   // --- Status ---
   IF #distance <= #tolerance THEN
       "HMI_Central_Shifter".CS_Status_Auto_Go_to_Des := 2;
   ELSIF #Drive_To_Pos THEN
       "HMI_Central_Shifter".CS_Status_Auto_Go_to_Des := 1;
   ELSE
       "HMI_Central_Shifter".CS_Status_Auto_Go_to_Des := 0;
   END_IF;



   // --- Granice bezpieczeństwa ---
   IF #Actual_Pos <= 0 THEN
       #Auto_Drive_Forward := FALSE;
       #Auto_Drive_Backward := FALSE;
       #Auto_Speed := 0.0;
       #DecelTimer.IN := FALSE;
       #RampActive := FALSE;
       #StopRampTimer.IN := FALSE;
   END_IF;
END_REGION
END_FUNCTION_BLOCK

FUNCTION_BLOCK "CentralShifter_SideShifters"   // FB17, LAD
{ S7_Optimized_Access := 'TRUE' }
// stored: MemoryReserve 100, SetENOAutomatically false
   VAR_INPUT
      In_Side_Drive_Pos : Bool;
      Position_CS : Int;
   END_VAR
   VAR_OUTPUT
      qLeftSide_in_Mid : Bool;
      qRightSide_in_Mid : Bool;
   END_VAR
   VAR
      Side_Hydraulic_CS_RL { S7_SetPoint := 'True'} : "Side_Hydraulic";
      Side_Hydraulic_CS_RR { S7_SetPoint := 'True'} : "Side_Hydraulic";
      Side_Driver_CS { S7_SetPoint := 'True'} : "Side_Driver";
      RL_Speed { S7_SetPoint := 'True'} : Int;
      RP_Speed : Int;
      CentralShifter_Side_Auto_Instance { S7_SetPoint := 'True'} : "CentralShifter_Side_Auto";
      SL_Auto_Speed { S7_SetPoint := 'True'} : Int;
      SR_Auto_Speed : Int;
      SL_Auto_Forward : Bool;
      SL_Auto_Backward : Bool;
      SR_Auto_Forward : Bool;
      SR_Auto_Backward : Bool;
      Sides_In_Position : Bool;
      Sides_In_H3_Pos : Bool;
      Sides_In_H5_Pos : Bool;
      Sides_In_CS_Pos : Bool;
      LightUp : Bool;
      LightMid : Bool;
      LightDown : Bool;
      SR_Error_Laser : Bool;
      SL_Error_Laser : Bool;
      Auto_Position_RL_Up : DInt;
      Auto_Position_RL_Mid : DInt;
      Auto_Position_RL_Down : DInt;
      Auto_Position_RR_Up : DInt;
      Auto_Position_RR_Mid : DInt;
      Auto_Position_RR_Down : DInt;
      Auto_Correction_RR : Int;
   END_VAR
   VAR RETAIN
      Stations : Array[7..13] of "CS_Sides_Stations";
   END_VAR
   VAR
      Status_Side_Go_H3 { S7_SetPoint := 'True'} : Int;
      Status_Side_Go_H5 : Int;
      Status_Side_Go_CS : Int;
      Auto_Hydraulic_Permission_H3 : Bool;
      Auto_Hydraulic_Permission_H5 : Bool;
      Auto_Hydraulic_Up_Timer { S7_SetPoint := 'True'} : TP_TIME;
      Auto_Hydraulic_Down_Timer { S7_SetPoint := 'True'} : TP_TIME;
      Station_H3_Empty : Bool;
      Station_H5_Empty : Bool;
      CS_R1_Sen_Up : Bool;
      CS_R1_Sen_Down : Bool;
      CS_R2_Sen_Up : Bool;
      CS_R2_Sen_Down : Bool;
      Auto_hyd_Up : Bool;
      Auto_hyd_Down : Bool;
      Hyd_Up_Status : Int;
      Hyd_Down_Status : Int;
      CS_RL_Error_Hyd : Bool;
      CS_RR_Error_Hyd : Bool;
      CS_Error_Hyd : Bool;
      CS_Error_Drive : Bool;
   END_VAR
   VAR CONSTANT
      Tolerance : Int := 60;
   END_VAR
   // Stations[7].RL_H3_Pos := 13516;
   // Stations[8].RL_H3_Pos := 13505;
   // Stations[9].RL_H3_Pos := 13520;
   // Stations[10].RL_H3_Pos := 13522;
   // Stations[11].RL_H3_Pos := 13526;
   // Stations[12].RL_H3_Pos := 13505;
   // Stations[13].RL_H3_Pos := 13500;
   // Stations[7].RR_H3_Pos := 13523;
   // Stations[8].RR_H3_Pos := 13495;
   // Stations[9].RR_H3_Pos := 13518;
   // Stations[10].RR_H3_Pos := 13527;
   // Stations[11].RR_H3_Pos := 13524;
   // Stations[12..13].RR_H3_Pos := 13525;
   // Stations[7].RL_Mid_Pos := 7915;
   // Stations[8].RL_Mid_Pos := 7910;
   // Stations[9].RL_Mid_Pos := 7933;
   // Stations[10].RL_Mid_Pos := 7928;
   // Stations[11].RL_Mid_Pos := 7937;
   // Stations[12].RL_Mid_Pos := 7932;
   // Stations[13].RL_Mid_Pos := 7916;
   // Stations[7].RR_Mid_Pos := 7925;
   // Stations[8].RR_Mid_Pos := 7895;
   // Stations[9].RR_Mid_Pos := 7922;
   // Stations[10].RR_Mid_Pos := 7935;
   // Stations[11].RR_Mid_Pos := 7926;
   // Stations[12].RR_Mid_Pos := 7932;
   // Stations[13].RR_Mid_Pos := 7939;
   // Stations[7].RL_H5_Pos := 1930;
   // Stations[8].RL_H5_Pos := 1917;
   // Stations[9].RL_H5_Pos := 1928;
   // Stations[10].RL_H5_Pos := 1929;
   // Stations[11].RL_H5_Pos := 1936;
   // Stations[12].RL_H5_Pos := 1924;
   // Stations[13].RL_H5_Pos := 1918;
   // Stations[7].RR_H5_Pos := 1929;
   // Stations[8].RR_H5_Pos := 1900;
   // Stations[9].RR_H5_Pos := 1921;
   // Stations[10].RR_H5_Pos := 1933;
   // Stations[11].RR_H5_Pos := 1928;
   // Stations[12].RR_H5_Pos := 1934;
   // Stations[13].RR_H5_Pos := 1915;
   // Stations[7].Correction := -20;
   // Stations[8].Correction := -15;
   // Stations[9].Correction := -5;
   // Stations[11].Correction := 0;
   // Stations[12].Correction := 10;
   // Stations[13].Correction := 15;
BEGIN

REGION Network 1: Hydraulic_RL
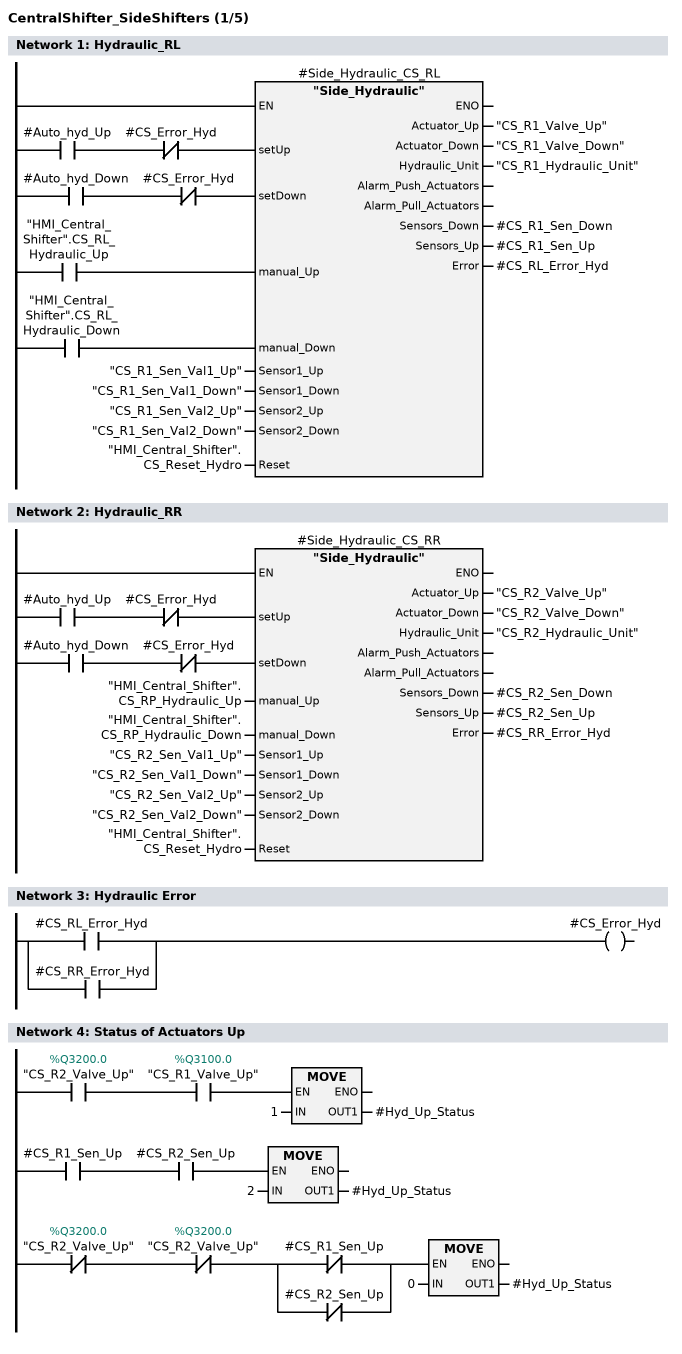
   RUNG wire#powerrail
      #Side_Hydraulic_CS_RL(setUp := wire#w1, setDown := wire#w2, manual_Up := wire#w3, manual_Down := wire#w4, Sensor1_Up := "CS_R1_Sen_Val1_Up", Sensor1_Down := "CS_R1_Sen_Val1_Down", Sensor2_Up := "CS_R1_Sen_Val2_Up", Sensor2_Down := "CS_R1_Sen_Val2_Down", Reset := "HMI_Central_Shifter".CS_Reset_Hydro, Actuator_Up => "CS_R1_Valve_Up", Actuator_Down => "CS_R1_Valve_Down", Hydraulic_Unit => "CS_R1_Hydraulic_Unit", Alarm_Push_Actuators =>, Alarm_Pull_Actuators =>, Sensors_Down => #CS_R1_Sen_Down, Sensors_Up => #CS_R1_Sen_Up, Error => #CS_RL_Error_Hyd)
   END_RUNG
   RUNG wire#powerrail
      Contact( #Auto_hyd_Up )
      I_Contact( #CS_Error_Hyd )
   END_RUNG wire#w1
   RUNG wire#powerrail
      Contact( #Auto_hyd_Down )
      I_Contact( #CS_Error_Hyd )
   END_RUNG wire#w2
   RUNG wire#powerrail
      Contact( "HMI_Central_Shifter".CS_RL_Hydraulic_Up )
   END_RUNG wire#w3
   RUNG wire#powerrail
      Contact( "HMI_Central_Shifter".CS_RL_Hydraulic_Down )
   END_RUNG wire#w4
   // the same network as SCL:
   #Side_Hydraulic_CS_RL(setUp := #Auto_hyd_Up AND NOT #CS_Error_Hyd,   // "Side_Hydraulic"
                         setDown := #Auto_hyd_Down AND NOT #CS_Error_Hyd,
                         manual_Up := "HMI_Central_Shifter".CS_RL_Hydraulic_Up,
                         manual_Down := "HMI_Central_Shifter".CS_RL_Hydraulic_Down,
                         Sensor1_Up := "CS_R1_Sen_Val1_Up",
                         Sensor1_Down := "CS_R1_Sen_Val1_Down",
                         Sensor2_Up := "CS_R1_Sen_Val2_Up",
                         Sensor2_Down := "CS_R1_Sen_Val2_Down",
                         Reset := "HMI_Central_Shifter".CS_Reset_Hydro,
                         Actuator_Up => "CS_R1_Valve_Up",
                         Actuator_Down => "CS_R1_Valve_Down",
                         Hydraulic_Unit => "CS_R1_Hydraulic_Unit",
                         Sensors_Down => #CS_R1_Sen_Down,
                         Sensors_Up => #CS_R1_Sen_Up,
                         Error => #CS_RL_Error_Hyd);
END_REGION

REGION Network 2: Hydraulic_RR
   RUNG wire#powerrail
      #Side_Hydraulic_CS_RR(setUp := wire#w1, setDown := wire#w2, manual_Up := "HMI_Central_Shifter".CS_RP_Hydraulic_Up, manual_Down := "HMI_Central_Shifter".CS_RP_Hydraulic_Down, Sensor1_Up := "CS_R2_Sen_Val1_Up", Sensor1_Down := "CS_R2_Sen_Val1_Down", Sensor2_Up := "CS_R2_Sen_Val2_Up", Sensor2_Down := "CS_R2_Sen_Val2_Down", Reset := "HMI_Central_Shifter".CS_Reset_Hydro, Actuator_Up => "CS_R2_Valve_Up", Actuator_Down => "CS_R2_Valve_Down", Hydraulic_Unit => "CS_R2_Hydraulic_Unit", Alarm_Push_Actuators =>, Alarm_Pull_Actuators =>, Sensors_Down => #CS_R2_Sen_Down, Sensors_Up => #CS_R2_Sen_Up, Error => #CS_RR_Error_Hyd)
   END_RUNG
   RUNG wire#powerrail
      Contact( #Auto_hyd_Up )
      I_Contact( #CS_Error_Hyd )
   END_RUNG wire#w1
   RUNG wire#powerrail
      Contact( #Auto_hyd_Down )
      I_Contact( #CS_Error_Hyd )
   END_RUNG wire#w2
   // the same network as SCL:
   #Side_Hydraulic_CS_RR(setUp := #Auto_hyd_Up AND NOT #CS_Error_Hyd,   // "Side_Hydraulic"
                         setDown := #Auto_hyd_Down AND NOT #CS_Error_Hyd,
                         manual_Up := "HMI_Central_Shifter".CS_RP_Hydraulic_Up,
                         manual_Down := "HMI_Central_Shifter".CS_RP_Hydraulic_Down,
                         Sensor1_Up := "CS_R2_Sen_Val1_Up",
                         Sensor1_Down := "CS_R2_Sen_Val1_Down",
                         Sensor2_Up := "CS_R2_Sen_Val2_Up",
                         Sensor2_Down := "CS_R2_Sen_Val2_Down",
                         Reset := "HMI_Central_Shifter".CS_Reset_Hydro,
                         Actuator_Up => "CS_R2_Valve_Up",
                         Actuator_Down => "CS_R2_Valve_Down",
                         Hydraulic_Unit => "CS_R2_Hydraulic_Unit",
                         Sensors_Down => #CS_R2_Sen_Down,
                         Sensors_Up => #CS_R2_Sen_Up,
                         Error => #CS_RR_Error_Hyd);
END_REGION

REGION Network 3: Hydraulic Error
   RUNG wire#powerrail
      Contact( #CS_RL_Error_Hyd )
      wire#w1
      Coil( #CS_Error_Hyd )
   END_RUNG
   RUNG wire#powerrail
      Contact( #CS_RR_Error_Hyd )
   END_RUNG wire#w1
   // the same network as SCL:
   #CS_Error_Hyd := #CS_RL_Error_Hyd OR #CS_RR_Error_Hyd;
END_REGION

REGION Network 4: Status of Actuators Up
   RUNG wire#powerrail
      Contact( "CS_R2_Valve_Up" )
      Contact( "CS_R1_Valve_Up" )
      Move(in := 1, out1 => #Hyd_Up_Status)
   END_RUNG
   RUNG wire#powerrail
      Contact( #CS_R1_Sen_Up )
      Contact( #CS_R2_Sen_Up )
      Move(in := 2, out1 => #Hyd_Up_Status)
   END_RUNG
   RUNG wire#powerrail
      I_Contact( "CS_R2_Valve_Up" )
      I_Contact( "CS_R2_Valve_Up" )
      wire#w1
      I_Contact( #CS_R1_Sen_Up )
      wire#w2
      Move(in := 0, out1 => #Hyd_Up_Status)
   END_RUNG
   RUNG wire#w1
      I_Contact( #CS_R2_Sen_Up )
   END_RUNG wire#w2
   // the same network as SCL:
   IF "CS_R2_Valve_Up" AND "CS_R1_Valve_Up" THEN #Hyd_Up_Status := 1; END_IF;
   IF #CS_R1_Sen_Up AND #CS_R2_Sen_Up THEN #Hyd_Up_Status := 2; END_IF;
   IF NOT "CS_R2_Valve_Up" AND NOT "CS_R2_Valve_Up" AND (NOT #CS_R1_Sen_Up OR NOT #CS_R2_Sen_Up) THEN
       #Hyd_Up_Status := 0;
   END_IF;
END_REGION

REGION Network 5: Status of Actuators Down
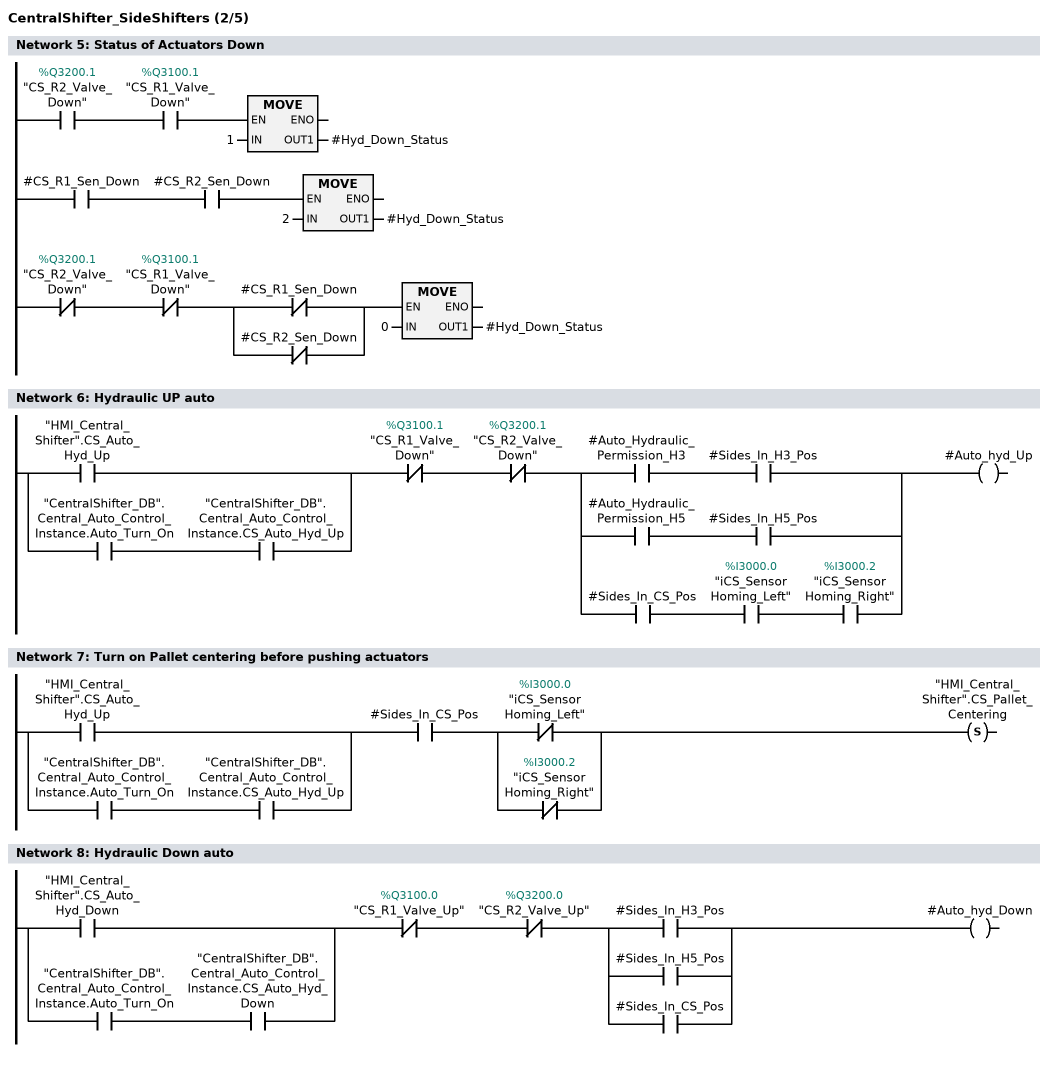
   RUNG wire#powerrail
      Contact( "CS_R2_Valve_Down" )
      Contact( "CS_R1_Valve_Down" )
      Move(in := 1, out1 => #Hyd_Down_Status)
   END_RUNG
   RUNG wire#powerrail
      Contact( #CS_R1_Sen_Down )
      Contact( #CS_R2_Sen_Down )
      Move(in := 2, out1 => #Hyd_Down_Status)
   END_RUNG
   RUNG wire#powerrail
      I_Contact( "CS_R2_Valve_Down" )
      I_Contact( "CS_R1_Valve_Down" )
      wire#w1
      I_Contact( #CS_R1_Sen_Down )
      wire#w2
      Move(in := 0, out1 => #Hyd_Down_Status)
   END_RUNG
   RUNG wire#w1
      I_Contact( #CS_R2_Sen_Down )
   END_RUNG wire#w2
   // the same network as SCL:
   IF "CS_R2_Valve_Down" AND "CS_R1_Valve_Down" THEN #Hyd_Down_Status := 1; END_IF;
   IF #CS_R1_Sen_Down AND #CS_R2_Sen_Down THEN #Hyd_Down_Status := 2; END_IF;
   IF NOT "CS_R2_Valve_Down" AND NOT "CS_R1_Valve_Down" AND (NOT #CS_R1_Sen_Down OR NOT #CS_R2_Sen_Down) THEN
       #Hyd_Down_Status := 0;
   END_IF;
END_REGION

REGION Network 6: Hydraulic UP auto
   RUNG wire#powerrail
      Contact( "HMI_Central_Shifter".CS_Auto_Hyd_Up )
      wire#w1
      I_Contact( "CS_R1_Valve_Down" )
      I_Contact( "CS_R2_Valve_Down" )
      wire#w2
      Contact( #Auto_Hydraulic_Permission_H3 )
      Contact( #Sides_In_H3_Pos )
      wire#w3
      Coil( #Auto_hyd_Up )
   END_RUNG
   RUNG wire#powerrail
      Contact( "CentralShifter_DB".Central_Auto_Control_Instance.Auto_Turn_On )
      Contact( "CentralShifter_DB".Central_Auto_Control_Instance.CS_Auto_Hyd_Up )
   END_RUNG wire#w1
   RUNG wire#w2
      Contact( #Auto_Hydraulic_Permission_H5 )
      Contact( #Sides_In_H5_Pos )
   END_RUNG wire#w3
   RUNG wire#w2
      Contact( #Sides_In_CS_Pos )
      Contact( "iCS_SensorHoming_Left" )
      Contact( "iCS_SensorHoming_Right" )
   END_RUNG wire#w3
   // the same network as SCL:
   #Auto_hyd_Up := ("HMI_Central_Shifter".CS_Auto_Hyd_Up OR ("CentralShifter_DB".Central_Auto_Control_Instance.Auto_Turn_On AND "CentralShifter_DB".Central_Auto_Control_Instance.CS_Auto_Hyd_Up)) AND NOT "CS_R1_Valve_Down" AND NOT "CS_R2_Valve_Down" AND ((#Auto_Hydraulic_Permission_H3 AND #Sides_In_H3_Pos) OR (#Auto_Hydraulic_Permission_H5 AND #Sides_In_H5_Pos) OR (#Sides_In_CS_Pos AND "iCS_SensorHoming_Left" AND "iCS_SensorHoming_Right"));
END_REGION

REGION Network 7: Turn on Pallet centering before pushing actuators
   RUNG wire#powerrail
      Contact( "HMI_Central_Shifter".CS_Auto_Hyd_Up )
      wire#w1
      Contact( #Sides_In_CS_Pos )
      wire#w2
      I_Contact( "iCS_SensorHoming_Left" )
      wire#w3
      S_Coil( "HMI_Central_Shifter".CS_Pallet_Centering )
   END_RUNG
   RUNG wire#powerrail
      Contact( "CentralShifter_DB".Central_Auto_Control_Instance.Auto_Turn_On )
      Contact( "CentralShifter_DB".Central_Auto_Control_Instance.CS_Auto_Hyd_Up )
   END_RUNG wire#w1
   RUNG wire#w2
      I_Contact( "iCS_SensorHoming_Right" )
   END_RUNG wire#w3
   // the same network as SCL:
   IF ("HMI_Central_Shifter".CS_Auto_Hyd_Up OR ("CentralShifter_DB".Central_Auto_Control_Instance.Auto_Turn_On AND "CentralShifter_DB".Central_Auto_Control_Instance.CS_Auto_Hyd_Up)) AND #Sides_In_CS_Pos AND (NOT "iCS_SensorHoming_Left" OR NOT "iCS_SensorHoming_Right") THEN
       "HMI_Central_Shifter".CS_Pallet_Centering := TRUE;
   END_IF;
END_REGION

REGION Network 8: Hydraulic Down auto
   RUNG wire#powerrail
      Contact( "HMI_Central_Shifter".CS_Auto_Hyd_Down )
      wire#w1
      I_Contact( "CS_R1_Valve_Up" )
      I_Contact( "CS_R2_Valve_Up" )
      wire#w2
      Contact( #Sides_In_H3_Pos )
      wire#w3
      Coil( #Auto_hyd_Down )
   END_RUNG
   RUNG wire#powerrail
      Contact( "CentralShifter_DB".Central_Auto_Control_Instance.Auto_Turn_On )
      Contact( "CentralShifter_DB".Central_Auto_Control_Instance.CS_Auto_Hyd_Down )
   END_RUNG wire#w1
   RUNG wire#w2
      Contact( #Sides_In_H5_Pos )
   END_RUNG wire#w3
   RUNG wire#w2
      Contact( #Sides_In_CS_Pos )
   END_RUNG wire#w3
   // the same network as SCL:
   #Auto_hyd_Down := ("HMI_Central_Shifter".CS_Auto_Hyd_Down OR ("CentralShifter_DB".Central_Auto_Control_Instance.Auto_Turn_On AND "CentralShifter_DB".Central_Auto_Control_Instance.CS_Auto_Hyd_Down)) AND NOT "CS_R1_Valve_Up" AND NOT "CS_R2_Valve_Up" AND (#Sides_In_H3_Pos OR #Sides_In_H5_Pos OR #Sides_In_CS_Pos);
END_REGION

REGION Network 9: Laser Error
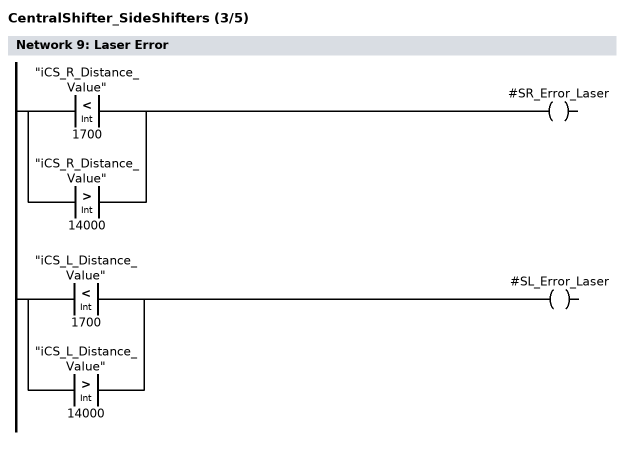
   RUNG wire#powerrail
      { S7_Templates := "SrcType := Int" } LT_Contact(in1 := "iCS_R_Distance_Value", in2 := 1700)
      wire#w1
      Coil( #SR_Error_Laser )
   END_RUNG
   RUNG wire#powerrail
      { S7_Templates := "SrcType := Int" } GT_Contact(in1 := "iCS_R_Distance_Value", in2 := 14000)
   END_RUNG wire#w1
   RUNG wire#powerrail
      { S7_Templates := "SrcType := Int" } LT_Contact(in1 := "iCS_L_Distance_Value", in2 := 1700)
      wire#w2
      Coil( #SL_Error_Laser )
   END_RUNG
   RUNG wire#powerrail
      { S7_Templates := "SrcType := Int" } GT_Contact(in1 := "iCS_L_Distance_Value", in2 := 14000)
   END_RUNG wire#w2
   // the same network as SCL:
   #SR_Error_Laser := ("iCS_R_Distance_Value" < 1700) OR ("iCS_R_Distance_Value" > 14000);
   #SL_Error_Laser := ("iCS_L_Distance_Value" < 1700) OR ("iCS_L_Distance_Value" > 14000);
END_REGION

REGION Network 10 (SCL): Setting SIDE positions by CS_POS
   CASE #Position_CS OF
       7..13:
           #Auto_Position_RL_Up := #Stations[#Position_CS].RL_H3_Pos;
           #Auto_Position_RR_Up := #Stations[#Position_CS].RR_H3_Pos;
           #Auto_Position_RL_Mid := #Stations[#Position_CS].RL_Mid_Pos;
           #Auto_Position_RR_Mid := #Stations[#Position_CS].RR_Mid_Pos;
           #Auto_Position_RL_Down := #Stations[#Position_CS].RL_H5_Pos;
           #Auto_Position_RR_Down := #Stations[#Position_CS].RR_H5_Pos;
           #Auto_Correction_RR := #Stations[#Position_CS].Correction;
       ELSE

           #Auto_Position_RL_Up := 0;
           #Auto_Position_RR_Up := 0;
           #Auto_Position_RL_Mid := 0;
           #Auto_Position_RR_Mid := 0;
           #Auto_Position_RL_Down := 0;
           #Auto_Position_RR_Down := 0;
           #Auto_Correction_RR := 0;
   END_CASE;
END_REGION

REGION Network 11 (SCL): Perform centering during hyd up
   CASE #Position_CS OF
       7..13:
           IF #Sides_In_H3_Pos AND ("HMI_Central_Shifter".CS_Auto_Hyd_Up OR ("CentralShifter_DB".Central_Auto_Control_Instance.Auto_Turn_On AND "CentralShifter_DB".Central_Auto_Control_Instance.CS_Auto_Hyd_Up)) AND NOT "System_To_Moving_Pallets_DB".Centering_Status[#Position_CS, 1] THEN
               "System_To_Moving_Pallets_DB".Centering_Perform[#Position_CS, 1] := 1;
           ELSIF #Sides_In_H5_Pos AND ("HMI_Central_Shifter".CS_Auto_Hyd_Up OR ("CentralShifter_DB".Central_Auto_Control_Instance.Auto_Turn_On AND "CentralShifter_DB".Central_Auto_Control_Instance.CS_Auto_Hyd_Up)) AND NOT "System_To_Moving_Pallets_DB".Centering_Status[#Position_CS, 3] THEN
               "System_To_Moving_Pallets_DB".Centering_Perform[#Position_CS, 3] := 1;
           END_IF;
   END_CASE;
END_REGION

REGION Network 12 (SCL): Permission to hyd up auto
   CASE #Position_CS OF
       7..13:
           IF "System_To_Moving_Pallets_DB".Centering_Status[#Position_CS, 1] THEN

               #Auto_Hydraulic_Permission_H3 := 1;
           ELSE
               #Auto_Hydraulic_Permission_H3 := 0;
           END_IF;

           IF "System_To_Moving_Pallets_DB".Centering_Status[#Position_CS, 3] THEN

               #Auto_Hydraulic_Permission_H5 := 1;
           ELSE
               #Auto_Hydraulic_Permission_H5 := 0;
           END_IF;

   END_CASE;
END_REGION

REGION Network 13 (SCL): Stations empty
   CASE #Position_CS OF
       7..13:
               #Station_H3_Empty := "Pallets_Stations".Stations[4, #Position_CS-3].IsEmpty;

               #Station_H5_Empty := "Pallets_Stations".Stations[2, #Position_CS-2].IsEmpty;

   END_CASE;
END_REGION

REGION Network 14: SIde Drivers
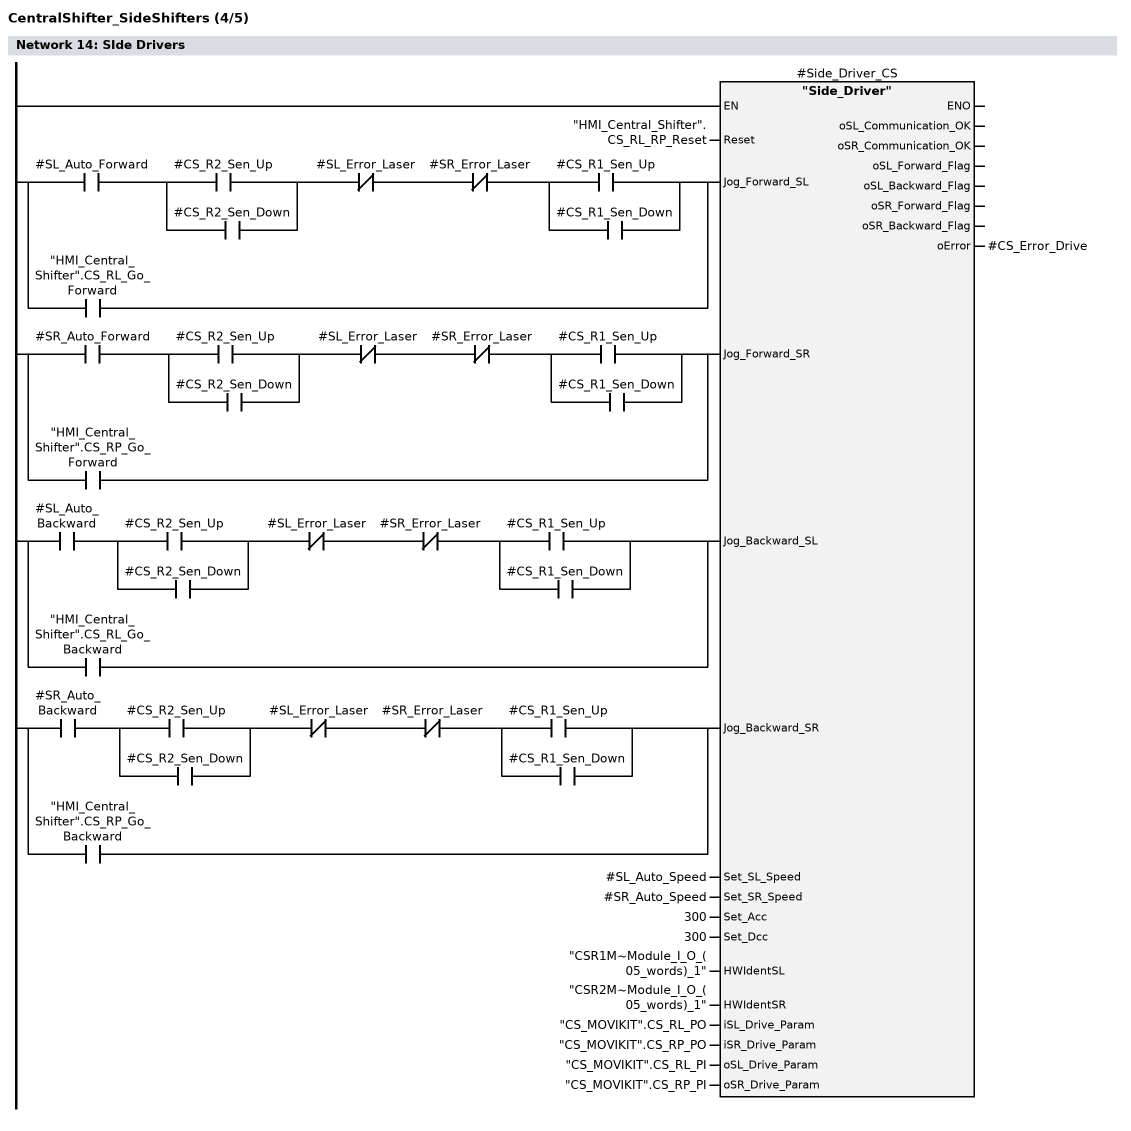
   RUNG wire#powerrail
      #Side_Driver_CS(Jog_Forward_SL := wire#w4, Jog_Forward_SR := wire#w8, Jog_Backward_SL := wire#w12, Jog_Backward_SR := wire#w16, Reset := "HMI_Central_Shifter".CS_RL_RP_Reset, Set_SL_Speed := #SL_Auto_Speed, Set_SR_Speed := #SR_Auto_Speed, Set_Acc := 300, Set_Dcc := 300, HWIdentSL := "CSR1M~Module_I_O_(05_words)_1", HWIdentSR := "CSR2M~Module_I_O_(05_words)_1", iSL_Drive_Param := "CS_MOVIKIT".CS_RL_PO, iSR_Drive_Param := "CS_MOVIKIT".CS_RP_PO, oSL_Drive_Param := "CS_MOVIKIT".CS_RL_PI, oSR_Drive_Param := "CS_MOVIKIT".CS_RP_PI, oSL_Communication_OK =>, oSR_Communication_OK =>, oSL_Forward_Flag =>, oSL_Backward_Flag =>, oSR_Forward_Flag =>, oSR_Backward_Flag =>, oError => #CS_Error_Drive)
   END_RUNG
   RUNG wire#powerrail
      Contact( #SL_Auto_Forward )
      wire#w1
      Contact( #CS_R2_Sen_Up )
      wire#w2
      I_Contact( #SL_Error_Laser )
      I_Contact( #SR_Error_Laser )
      wire#w3
      Contact( #CS_R1_Sen_Up )
   END_RUNG wire#w4
   RUNG wire#w1
      Contact( #CS_R2_Sen_Down )
   END_RUNG wire#w2
   RUNG wire#w3
      Contact( #CS_R1_Sen_Down )
   END_RUNG wire#w4
   RUNG wire#powerrail
      Contact( "HMI_Central_Shifter".CS_RL_Go_Forward )
   END_RUNG wire#w4
   RUNG wire#powerrail
      Contact( #SR_Auto_Forward )
      wire#w5
      Contact( #CS_R2_Sen_Up )
      wire#w6
      I_Contact( #SL_Error_Laser )
      I_Contact( #SR_Error_Laser )
      wire#w7
      Contact( #CS_R1_Sen_Up )
   END_RUNG wire#w8
   RUNG wire#w5
      Contact( #CS_R2_Sen_Down )
   END_RUNG wire#w6
   RUNG wire#w7
      Contact( #CS_R1_Sen_Down )
   END_RUNG wire#w8
   RUNG wire#powerrail
      Contact( "HMI_Central_Shifter".CS_RP_Go_Forward )
   END_RUNG wire#w8
   RUNG wire#powerrail
      Contact( #SL_Auto_Backward )
      wire#w9
      Contact( #CS_R2_Sen_Up )
      wire#w10
      I_Contact( #SL_Error_Laser )
      I_Contact( #SR_Error_Laser )
      wire#w11
      Contact( #CS_R1_Sen_Up )
   END_RUNG wire#w12
   RUNG wire#w9
      Contact( #CS_R2_Sen_Down )
   END_RUNG wire#w10
   RUNG wire#w11
      Contact( #CS_R1_Sen_Down )
   END_RUNG wire#w12
   RUNG wire#powerrail
      Contact( "HMI_Central_Shifter".CS_RL_Go_Backward )
   END_RUNG wire#w12
   RUNG wire#powerrail
      Contact( #SR_Auto_Backward )
      wire#w13
      Contact( #CS_R2_Sen_Up )
      wire#w14
      I_Contact( #SL_Error_Laser )
      I_Contact( #SR_Error_Laser )
      wire#w15
      Contact( #CS_R1_Sen_Up )
   END_RUNG wire#w16
   RUNG wire#w13
      Contact( #CS_R2_Sen_Down )
   END_RUNG wire#w14
   RUNG wire#w15
      Contact( #CS_R1_Sen_Down )
   END_RUNG wire#w16
   RUNG wire#powerrail
      Contact( "HMI_Central_Shifter".CS_RP_Go_Backward )
   END_RUNG wire#w16
   // the same network as SCL:
   #Side_Driver_CS(Reset := "HMI_Central_Shifter".CS_RL_RP_Reset,   // "Side_Driver"
                   Jog_Forward_SL := (#SL_Auto_Forward AND (#CS_R2_Sen_Up OR #CS_R2_Sen_Down) AND NOT #SL_Error_Laser AND NOT #SR_Error_Laser AND (#CS_R1_Sen_Up OR #CS_R1_Sen_Down)) OR "HMI_Central_Shifter".CS_RL_Go_Forward,
                   Jog_Forward_SR := (#SR_Auto_Forward AND (#CS_R2_Sen_Up OR #CS_R2_Sen_Down) AND NOT #SL_Error_Laser AND NOT #SR_Error_Laser AND (#CS_R1_Sen_Up OR #CS_R1_Sen_Down)) OR "HMI_Central_Shifter".CS_RP_Go_Forward,
                   Jog_Backward_SL := (#SL_Auto_Backward AND (#CS_R2_Sen_Up OR #CS_R2_Sen_Down) AND NOT #SL_Error_Laser AND NOT #SR_Error_Laser AND (#CS_R1_Sen_Up OR #CS_R1_Sen_Down)) OR "HMI_Central_Shifter".CS_RL_Go_Backward,
                   Jog_Backward_SR := (#SR_Auto_Backward AND (#CS_R2_Sen_Up OR #CS_R2_Sen_Down) AND NOT #SL_Error_Laser AND NOT #SR_Error_Laser AND (#CS_R1_Sen_Up OR #CS_R1_Sen_Down)) OR "HMI_Central_Shifter".CS_RP_Go_Backward,
                   Set_SL_Speed := #SL_Auto_Speed,
                   Set_SR_Speed := #SR_Auto_Speed,
                   Set_Acc := 300,
                   Set_Dcc := 300,
                   HWIdentSL := "CSR1M~Module_I_O_(05_words)_1",
                   HWIdentSR := "CSR2M~Module_I_O_(05_words)_1",
                   iSL_Drive_Param := "CS_MOVIKIT".CS_RL_PO,
                   iSR_Drive_Param := "CS_MOVIKIT".CS_RP_PO,
                   oSL_Drive_Param := "CS_MOVIKIT".CS_RL_PI,
                   oSR_Drive_Param := "CS_MOVIKIT".CS_RP_PI,
                   oError => #CS_Error_Drive);
END_REGION

REGION Network 15 (SCL): Limit positions of Sides
   IF #Auto_Position_RL_Down > 14000 THEN
       #Auto_Position_RL_Down := 14000;
   ELSIF #Auto_Position_RL_Down < 1800 THEN
       #Auto_Position_RL_Down := 1800;
   END_IF;

   IF #Auto_Position_RL_Up > 14000 THEN
       #Auto_Position_RL_Up := 14000;
   ELSIF #Auto_Position_RL_Up < 1800 THEN
       #Auto_Position_RL_Up := 1800;
   END_IF;

   IF #Auto_Position_RR_Down > 14000 THEN
       #Auto_Position_RR_Down := 14000;
   ELSIF #Auto_Position_RR_Down < 1800 THEN
       #Auto_Position_RR_Down := 1800;
   END_IF;

   IF #Auto_Position_RR_Up > 14000 THEN
       #Auto_Position_RR_Up := 14000;
   ELSIF #Auto_Position_RR_Up < 1800 THEN
       #Auto_Position_RR_Up := 1800;
   END_IF;
END_REGION

REGION Network 16: CS Side Auto
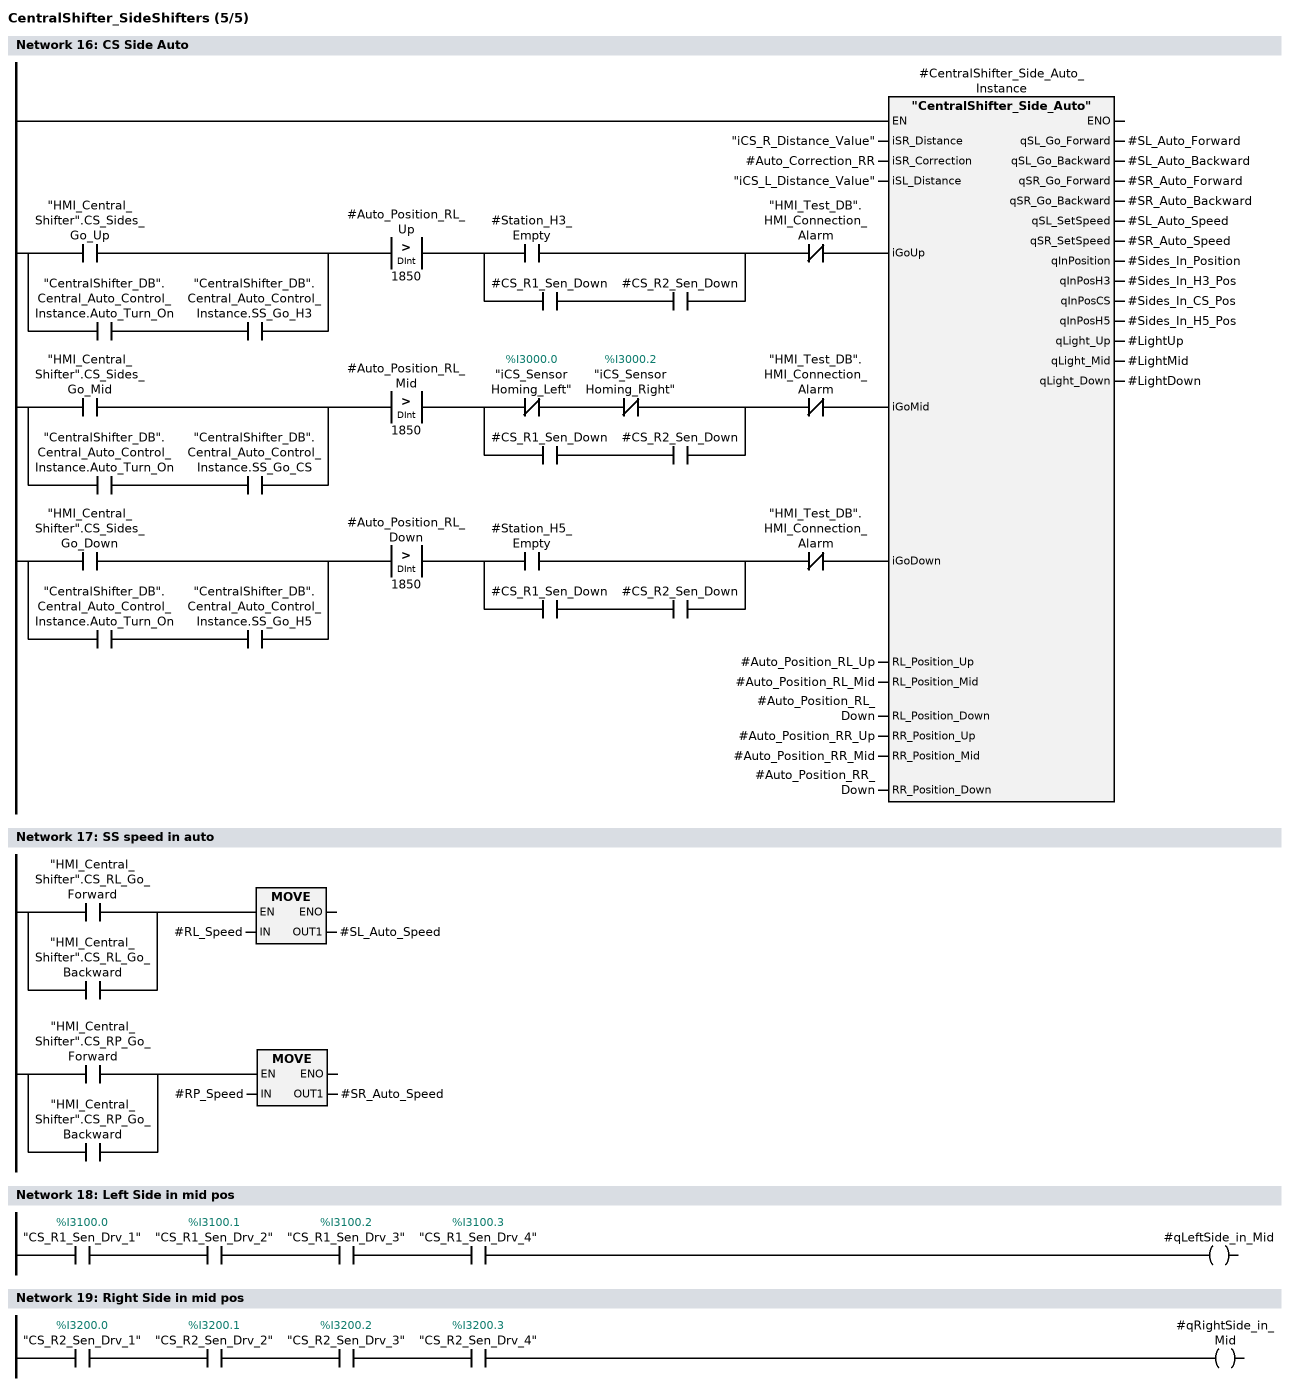
   RUNG wire#powerrail
      #CentralShifter_Side_Auto_Instance(iGoUp := wire#w4, iGoMid := wire#w8, iGoDown := wire#w12, iSR_Distance := "iCS_R_Distance_Value", iSR_Correction := #Auto_Correction_RR, iSL_Distance := "iCS_L_Distance_Value", RL_Position_Up := #Auto_Position_RL_Up, RL_Position_Mid := #Auto_Position_RL_Mid, RL_Position_Down := #Auto_Position_RL_Down, RR_Position_Up := #Auto_Position_RR_Up, RR_Position_Mid := #Auto_Position_RR_Mid, RR_Position_Down := #Auto_Position_RR_Down, qSL_Go_Forward => #SL_Auto_Forward, qSL_Go_Backward => #SL_Auto_Backward, qSR_Go_Forward => #SR_Auto_Forward, qSR_Go_Backward => #SR_Auto_Backward, qSL_SetSpeed => #SL_Auto_Speed, qSR_SetSpeed => #SR_Auto_Speed, qInPosition => #Sides_In_Position, qInPosH3 => #Sides_In_H3_Pos, qInPosCS => #Sides_In_CS_Pos, qInPosH5 => #Sides_In_H5_Pos, qLight_Up => #LightUp, qLight_Mid => #LightMid, qLight_Down => #LightDown)
   END_RUNG
   RUNG wire#powerrail
      Contact( "HMI_Central_Shifter".CS_Sides_Go_Up )
      wire#w1
      { S7_Templates := "SrcType := DInt" } GT_Contact(in1 := #Auto_Position_RL_Up, in2 := 1850)
      wire#w2
      Contact( #Station_H3_Empty )
      wire#w3
      I_Contact( "HMI_Test_DB".HMI_Connection_Alarm )
   END_RUNG wire#w4
   RUNG wire#powerrail
      Contact( "CentralShifter_DB".Central_Auto_Control_Instance.Auto_Turn_On )
      Contact( "CentralShifter_DB".Central_Auto_Control_Instance.SS_Go_H3 )
   END_RUNG wire#w1
   RUNG wire#w2
      Contact( #CS_R1_Sen_Down )
      Contact( #CS_R2_Sen_Down )
   END_RUNG wire#w3
   RUNG wire#powerrail
      Contact( "HMI_Central_Shifter".CS_Sides_Go_Mid )
      wire#w5
      { S7_Templates := "SrcType := DInt" } GT_Contact(in1 := #Auto_Position_RL_Mid, in2 := 1850)
      wire#w6
      I_Contact( "iCS_SensorHoming_Left" )
      I_Contact( "iCS_SensorHoming_Right" )
      wire#w7
      I_Contact( "HMI_Test_DB".HMI_Connection_Alarm )
   END_RUNG wire#w8
   RUNG wire#powerrail
      Contact( "CentralShifter_DB".Central_Auto_Control_Instance.Auto_Turn_On )
      Contact( "CentralShifter_DB".Central_Auto_Control_Instance.SS_Go_CS )
   END_RUNG wire#w5
   RUNG wire#w6
      Contact( #CS_R1_Sen_Down )
      Contact( #CS_R2_Sen_Down )
   END_RUNG wire#w7
   RUNG wire#powerrail
      Contact( "HMI_Central_Shifter".CS_Sides_Go_Down )
      wire#w9
      { S7_Templates := "SrcType := DInt" } GT_Contact(in1 := #Auto_Position_RL_Down, in2 := 1850)
      wire#w10
      Contact( #Station_H5_Empty )
      wire#w11
      I_Contact( "HMI_Test_DB".HMI_Connection_Alarm )
   END_RUNG wire#w12
   RUNG wire#powerrail
      Contact( "CentralShifter_DB".Central_Auto_Control_Instance.Auto_Turn_On )
      Contact( "CentralShifter_DB".Central_Auto_Control_Instance.SS_Go_H5 )
   END_RUNG wire#w9
   RUNG wire#w10
      Contact( #CS_R1_Sen_Down )
      Contact( #CS_R2_Sen_Down )
   END_RUNG wire#w11
   // the same network as SCL:
   #CentralShifter_Side_Auto_Instance(iSR_Distance := "iCS_R_Distance_Value",   // "CentralShifter_Side_Auto"
                           iSR_Correction := #Auto_Correction_RR,
                           iSL_Distance := "iCS_L_Distance_Value",
                           iGoUp := ("HMI_Central_Shifter".CS_Sides_Go_Up OR ("CentralShifter_DB".Central_Auto_Control_Instance.Auto_Turn_On AND "CentralShifter_DB".Central_Auto_Control_Instance.SS_Go_H3)) AND (#Auto_Position_RL_Up > 1850) AND (#Station_H3_Empty OR (#CS_R1_Sen_Down AND #CS_R2_Sen_Down)) AND NOT "HMI_Test_DB".HMI_Connection_Alarm,
                           iGoMid := ("HMI_Central_Shifter".CS_Sides_Go_Mid OR ("CentralShifter_DB".Central_Auto_Control_Instance.Auto_Turn_On AND "CentralShifter_DB".Central_Auto_Control_Instance.SS_Go_CS)) AND (#Auto_Position_RL_Mid > 1850) AND ((NOT "iCS_SensorHoming_Left" AND NOT "iCS_SensorHoming_Right") OR (#CS_R1_Sen_Down AND #CS_R2_Sen_Down)) AND NOT "HMI_Test_DB".HMI_Connection_Alarm,
                           iGoDown := ("HMI_Central_Shifter".CS_Sides_Go_Down OR ("CentralShifter_DB".Central_Auto_Control_Instance.Auto_Turn_On AND "CentralShifter_DB".Central_Auto_Control_Instance.SS_Go_H5)) AND (#Auto_Position_RL_Down > 1850) AND (#Station_H5_Empty OR (#CS_R1_Sen_Down AND #CS_R2_Sen_Down)) AND NOT "HMI_Test_DB".HMI_Connection_Alarm,
                           RL_Position_Up := #Auto_Position_RL_Up,
                           RL_Position_Mid := #Auto_Position_RL_Mid,
                           RL_Position_Down := #Auto_Position_RL_Down,
                           RR_Position_Up := #Auto_Position_RR_Up,
                           RR_Position_Mid := #Auto_Position_RR_Mid,
                           RR_Position_Down := #Auto_Position_RR_Down,
                           qSL_Go_Forward => #SL_Auto_Forward,
                           qSL_Go_Backward => #SL_Auto_Backward,
                           qSR_Go_Forward => #SR_Auto_Forward,
                           qSR_Go_Backward => #SR_Auto_Backward,
                           qSL_SetSpeed => #SL_Auto_Speed,
                           qSR_SetSpeed => #SR_Auto_Speed,
                           qInPosition => #Sides_In_Position,
                           qInPosH3 => #Sides_In_H3_Pos,
                           qInPosCS => #Sides_In_CS_Pos,
                           qInPosH5 => #Sides_In_H5_Pos,
                           qLight_Up => #LightUp,
                           qLight_Mid => #LightMid,
                           qLight_Down => #LightDown);
END_REGION

REGION Network 17: SS speed in auto
   RUNG wire#powerrail
      Contact( "HMI_Central_Shifter".CS_RL_Go_Forward )
      wire#w1
      Move(in := #RL_Speed, out1 => #SL_Auto_Speed)
   END_RUNG
   RUNG wire#powerrail
      Contact( "HMI_Central_Shifter".CS_RL_Go_Backward )
   END_RUNG wire#w1
   RUNG wire#powerrail
      Contact( "HMI_Central_Shifter".CS_RP_Go_Forward )
      wire#w2
      Move(in := #RP_Speed, out1 => #SR_Auto_Speed)
   END_RUNG
   RUNG wire#powerrail
      Contact( "HMI_Central_Shifter".CS_RP_Go_Backward )
   END_RUNG wire#w2
   // the same network as SCL:
   IF "HMI_Central_Shifter".CS_RL_Go_Forward OR "HMI_Central_Shifter".CS_RL_Go_Backward THEN
       #SL_Auto_Speed := #RL_Speed;
   END_IF;
   IF "HMI_Central_Shifter".CS_RP_Go_Forward OR "HMI_Central_Shifter".CS_RP_Go_Backward THEN
       #SR_Auto_Speed := #RP_Speed;
   END_IF;
END_REGION

REGION Network 18: Left Side in mid pos
   RUNG wire#powerrail
      Contact( "CS_R1_Sen_Drv_1" )
      Contact( "CS_R1_Sen_Drv_2" )
      Contact( "CS_R1_Sen_Drv_3" )
      Contact( "CS_R1_Sen_Drv_4" )
      Coil( #qLeftSide_in_Mid )
   END_RUNG
   // the same network as SCL:
   #qLeftSide_in_Mid := "CS_R1_Sen_Drv_1" AND "CS_R1_Sen_Drv_2" AND "CS_R1_Sen_Drv_3" AND "CS_R1_Sen_Drv_4";
END_REGION

REGION Network 19: Right Side in mid pos
   RUNG wire#powerrail
      Contact( "CS_R2_Sen_Drv_1" )
      Contact( "CS_R2_Sen_Drv_2" )
      Contact( "CS_R2_Sen_Drv_3" )
      Contact( "CS_R2_Sen_Drv_4" )
      Coil( #qRightSide_in_Mid )
   END_RUNG
   // the same network as SCL:
   #qRightSide_in_Mid := "CS_R2_Sen_Drv_1" AND "CS_R2_Sen_Drv_2" AND "CS_R2_Sen_Drv_3" AND "CS_R2_Sen_Drv_4";
END_REGION

REGION Network 20 (SCL): Status - go to destinations
           IF "HMI_Central_Shifter".CS_Sides_Go_Up AND NOT #Sides_In_H3_Pos AND #In_Side_Drive_Pos THEN
               #Status_Side_Go_H3 := 1;
           ELSIF #Sides_In_H3_Pos THEN
               #Status_Side_Go_H3 := 2;
           ELSE
               #Status_Side_Go_H3 := 0;
           END_IF;

           IF "HMI_Central_Shifter".CS_Sides_Go_Down AND NOT #Sides_In_H5_Pos AND #In_Side_Drive_Pos THEN
               #Status_Side_Go_H5 := 1;
           ELSIF #Sides_In_H5_Pos THEN
               #Status_Side_Go_H5 := 2;
           ELSE
               #Status_Side_Go_H5 := 0;
           END_IF;

           IF "HMI_Central_Shifter".CS_Sides_Go_Mid AND NOT #Sides_In_CS_Pos AND #In_Side_Drive_Pos THEN
               #Status_Side_Go_CS := 1;
           ELSIF #Sides_In_CS_Pos THEN
               #Status_Side_Go_CS := 2;
           ELSE
               #Status_Side_Go_CS := 0;
           END_IF;
END_REGION
END_FUNCTION_BLOCK

FUNCTION_BLOCK "CentralShifter_Side_Auto"
{ S7_Optimized_Access := 'TRUE' }
VERSION : 0.1
   VAR_INPUT 
      iSR_Distance : Int;
      iSR_Correction : Int;
      iSL_Distance : Int;
      iGoUp : Bool;
      iGoMid : Bool;
      iGoDown : Bool;
      RL_Position_Up : DInt;
      RL_Position_Mid : DInt;
      RL_Position_Down : DInt;
      RR_Position_Up : DInt;
      RR_Position_Mid : DInt;
      RR_Position_Down : DInt;
   END_VAR

   VAR_OUTPUT 
      qSL_Go_Forward : Bool;
      qSL_Go_Backward : Bool;
      qSR_Go_Forward : Bool;
      qSR_Go_Backward : Bool;
      qSL_SetSpeed : Int;
      qSR_SetSpeed : Int;
      qInPosition : Bool;
      qInPosH3 : Bool;
      qInPosCS : Bool;
      qInPosH5 : Bool;
      qLight_Up : Bool;
      qLight_Mid : Bool;
      qLight_Down : Bool;
   END_VAR

   VAR 
      distanceSL_SR : DInt;
      SR_Correct_Distance : DInt;
      moveActive : Bool;
      targetPosRL : DInt;
      targetPosRR : DInt;
      distanceToTargetSL : DInt;
      distanceToTargetSR : DInt;
      Delta : Real;
   END_VAR

   VAR CONSTANT 
      Tolerance : Int := 2;
      Tolerance_Hydro : Int := 7;
      Tolerance_Light : Int := 10;
      DistanceSlowZone : Int := 300;
      K : Real := 1.5;
      Tolerance_CS : Int := 25;
   END_VAR


BEGIN
	// Reset komend ruchu
	#qSL_Go_Forward := FALSE;
	#qSL_Go_Backward := FALSE;
	#qSR_Go_Forward := FALSE;
	#qSR_Go_Backward := FALSE;
	
	#SR_Correct_Distance := #iSR_Correction + #iSR_Distance;
	#distanceSL_SR := #SR_Correct_Distance - #iSL_Distance;
	
	
	// --- Miganie tylko gdy przycisk TRZYMANY i moveActive ---
	IF #moveActive AND "Clock_2Hz" THEN
	    IF #iGoDown THEN
	        #qLight_Down := 1;
	    ELSE
	        #qLight_Down := 0;
	    END_IF;
	    IF #iGoMid THEN
	        #qLight_Mid := 1;
	    ELSE
	        #qLight_Mid := 0;
	    END_IF;
	    IF #iGoUp THEN
	        #qLight_Up := 1;
	    ELSE
	        #qLight_Up := 0;
	    END_IF;
	ELSE
	    // Gdy nie ma ruchu — zgaś lampki
	    #qLight_Down:= 0;
	    #qLight_Mid := 0;
	    #qLight_Up := 0;
	END_IF;
	
	
	// --- Obsługa dynamicznego wyboru celu ---
	IF #iGoUp THEN
	    #targetPosRL := #RL_Position_Up;
	    #targetPosRR := #RR_Position_Up;
	    #moveActive := TRUE;
	ELSIF #iGoMid THEN
	    #targetPosRL := #RL_Position_Mid;
	    #targetPosRR := #RR_Position_Mid;
	    #moveActive := TRUE;
	ELSIF #iGoDown THEN
	    #targetPosRL := #RL_Position_Down;
	    #targetPosRR := #RR_Position_Down;
	    #moveActive := TRUE;
	ELSE
	    // Żaden przycisk nie trzymany — przerwij ruch
	    #moveActive := FALSE;
	END_IF;
	
	IF NOT "Data_From_Safety".Safety_Active THEN
	    #moveActive := 0;
	    ;
	END_IF;
	
	// --- Jeśli ruch aktywny ---
	IF #moveActive THEN
	    // --- SL (główny) ---
	    #distanceToTargetSL := ABS(#iSL_Distance - #targetPosRL);
	    #distanceToTargetSR := ABS(#SR_Correct_Distance - #targetPosRR);
	    
	    IF #distanceToTargetSL > #Tolerance THEN
	        IF #iSL_Distance > #targetPosRL THEN
	            #qSL_Go_Forward := FALSE;
	            #qSL_Go_Backward := TRUE;
	        ELSE
	            #qSL_Go_Forward := TRUE;
	            #qSL_Go_Backward := FALSE;
	        END_IF;
	        
	        IF #distanceToTargetSL <= #DistanceSlowZone THEN
	            #qSL_SetSpeed := 300;
	        ELSE
	            #qSL_SetSpeed := 1000;
	        END_IF;
	        
	    ELSE
	        #qSL_Go_Forward := FALSE;
	        #qSL_Go_Backward := FALSE;
	        #qSL_SetSpeed := 0;
	        #moveActive := FALSE;
	    END_IF;
	    
	    // --- SR (podąża) ---
	    #distanceSL_SR := #SR_Correct_Distance - #iSL_Distance;
	    //#absDelta := ABS(#distanceSL_SR);
	    // IF #distanceToTargetSL > #Tolerance THEN
	    
	    IF #distanceToTargetSR > #Tolerance THEN
	        IF #SR_Correct_Distance > #targetPosRR THEN
	            #qSR_Go_Forward := FALSE;
	            #qSR_Go_Backward := TRUE;
	        ELSE
	            #qSR_Go_Forward := TRUE;
	            #qSR_Go_Backward := FALSE;
	        END_IF;
	    END_IF;
	    
	    // Kierunek SR = kierunek SL
	    // #qSR_Go_Forward := #qSL_Go_Forward;
	    //#qSR_Go_Backward := #qSL_Go_Backward;
	    
	    // Korekcja prędkości
	    #Delta := #distanceSL_SR * #K;
	    IF #Delta > 1000 THEN
	        #Delta := 1000;
	    ELSIF #Delta < -1000 THEN
	        #Delta := -1000;
	    END_IF;
	    //zamien znaki
	    IF #qSR_Go_Forward THEN
	        #qSR_SetSpeed := #qSL_SetSpeed - #Delta;
	    ELSIF #qSR_Go_Backward THEN
	        #qSR_SetSpeed := #qSL_SetSpeed + #Delta;
	    END_IF;
	    
	    // Ograniczenia
	    IF #qSR_SetSpeed > 1500 THEN
	        #qSR_SetSpeed := 1500;
	    ELSIF #qSR_SetSpeed < 200 THEN
	        #qSR_SetSpeed := 200;
	    END_IF;
	    
	    // END_IF;
	END_IF;
	
	#qInPosition := FALSE;
	#qInPosH3 := FALSE;
	#qInPosCS := FALSE;
	#qInPosH5 := FALSE;
	
	// dolna
	IF (ABS(#iSL_Distance - #RL_Position_Down) <= #Tolerance_Hydro AND ABS(#SR_Correct_Distance - #RR_Position_Down) <= #Tolerance_Hydro) THEN
	    #qInPosition := TRUE;
	    #qInPosH5 := TRUE;
	    
	// cs
	ELSIF (ABS(#iSL_Distance - #RL_Position_Mid) <= #Tolerance_Hydro AND ABS(#SR_Correct_Distance - #RR_Position_Mid) <= #Tolerance_Hydro) THEN
	    #qInPosition := TRUE;
	    #qInPosCS := TRUE;
	    
	// górna
	ELSIF (ABS(#iSL_Distance - #RL_Position_Up) <= #Tolerance_Hydro AND ABS(#SR_Correct_Distance - #RR_Position_Up) <= #Tolerance_Hydro) THEN
	    #qInPosition := TRUE;
	    #qInPosH3 := TRUE;
	END_IF;
	
	
	
	IF (ABS(#iSL_Distance - #RL_Position_Down) <= #Tolerance_Light AND ABS(#SR_Correct_Distance - #RL_Position_Down) <= #Tolerance_Light) THEN
	    #qLight_Down := 1;
	ELSIF (ABS(#iSL_Distance - #RL_Position_Mid) <= #Tolerance_Light AND ABS(#SR_Correct_Distance - #RL_Position_Mid) <= #Tolerance_Light) THEN
	    #qLight_Mid := 1;
	ELSIF (ABS(#iSL_Distance - #RL_Position_Up) <= #Tolerance_Light AND ABS(#SR_Correct_Distance - #RL_Position_Up) <= #Tolerance_Light) THEN
	    #qLight_Up := 1;
	END_IF;
	
END_FUNCTION_BLOCK

FUNCTION_BLOCK "CentralShifter_Move_Pallets"   // FB19, LAD
{ S7_Optimized_Access := 'TRUE' }
// stored: MemoryReserve 100, SetENOAutomatically false
   VAR
      Motor_Driver_Instance { S7_SetPoint := 'True'} : "Side_Driver";
      Speed : Int := 400;
      Auto_Go_Left : Bool;
      Auto_Go_Right : Bool;
      CSM1_Comm_ok : Bool;
      CSM2_Comm_ok : Bool;
      prevCentering : Bool;
      tCenteringTimer : TON_TIME;
   END_VAR
   VAR_TEMP
      "czujnik lewy" : Bool;
      "czujnik prawy" : Bool;
   END_VAR
BEGIN

REGION Network 1
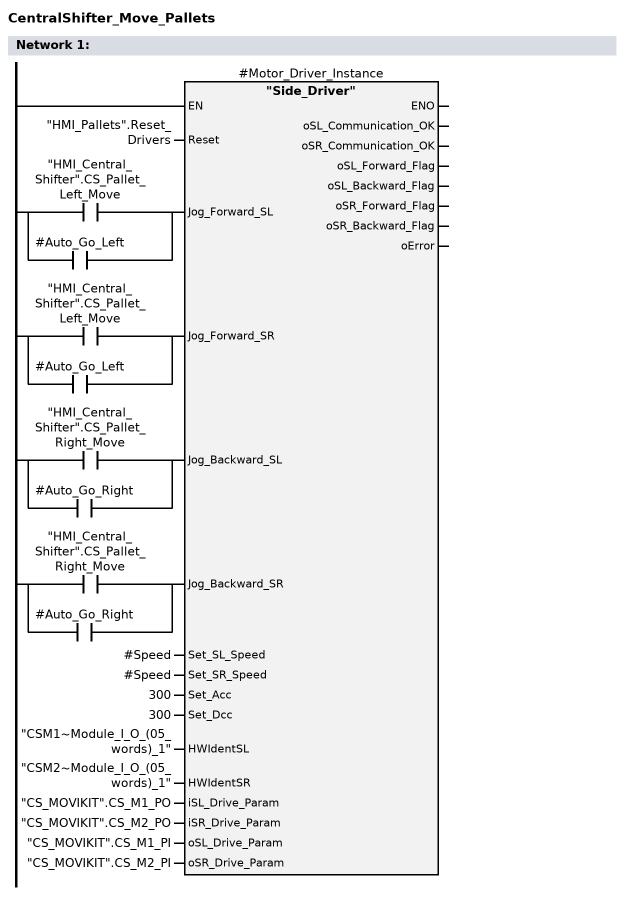
   RUNG wire#powerrail
      #Motor_Driver_Instance(Jog_Forward_SL := wire#w1, Jog_Forward_SR := wire#w2, Jog_Backward_SL := wire#w3, Jog_Backward_SR := wire#w4, Reset := "HMI_Pallets".Reset_Drivers, Set_SL_Speed := #Speed, Set_SR_Speed := #Speed, Set_Acc := 300, Set_Dcc := 300, HWIdentSL := "CSM1~Module_I_O_(05_words)_1", HWIdentSR := "CSM2~Module_I_O_(05_words)_1", iSL_Drive_Param := "CS_MOVIKIT".CS_M1_PO, iSR_Drive_Param := "CS_MOVIKIT".CS_M2_PO, oSL_Drive_Param := "CS_MOVIKIT".CS_M1_PI, oSR_Drive_Param := "CS_MOVIKIT".CS_M2_PI, oSL_Communication_OK =>, oSR_Communication_OK =>, oSL_Forward_Flag =>, oSL_Backward_Flag =>, oSR_Forward_Flag =>, oSR_Backward_Flag =>, oError =>)
   END_RUNG
   RUNG wire#powerrail
      Contact( "HMI_Central_Shifter".CS_Pallet_Left_Move )
   END_RUNG wire#w1
   RUNG wire#powerrail
      Contact( #Auto_Go_Left )
   END_RUNG wire#w1
   RUNG wire#powerrail
      Contact( "HMI_Central_Shifter".CS_Pallet_Left_Move )
   END_RUNG wire#w2
   RUNG wire#powerrail
      Contact( #Auto_Go_Left )
   END_RUNG wire#w2
   RUNG wire#powerrail
      Contact( "HMI_Central_Shifter".CS_Pallet_Right_Move )
   END_RUNG wire#w3
   RUNG wire#powerrail
      Contact( #Auto_Go_Right )
   END_RUNG wire#w3
   RUNG wire#powerrail
      Contact( "HMI_Central_Shifter".CS_Pallet_Right_Move )
   END_RUNG wire#w4
   RUNG wire#powerrail
      Contact( #Auto_Go_Right )
   END_RUNG wire#w4
   // the same network as SCL:
   #Motor_Driver_Instance(Reset := "HMI_Pallets".Reset_Drivers,   // "Side_Driver"
                          Jog_Forward_SL := "HMI_Central_Shifter".CS_Pallet_Left_Move OR #Auto_Go_Left,
                          Jog_Forward_SR := "HMI_Central_Shifter".CS_Pallet_Left_Move OR #Auto_Go_Left,
                          Jog_Backward_SL := "HMI_Central_Shifter".CS_Pallet_Right_Move OR #Auto_Go_Right,
                          Jog_Backward_SR := "HMI_Central_Shifter".CS_Pallet_Right_Move OR #Auto_Go_Right,
                          Set_SL_Speed := #Speed,
                          Set_SR_Speed := #Speed,
                          Set_Acc := 300,
                          Set_Dcc := 300,
                          HWIdentSL := "CSM1~Module_I_O_(05_words)_1",
                          HWIdentSR := "CSM2~Module_I_O_(05_words)_1",
                          iSL_Drive_Param := "CS_MOVIKIT".CS_M1_PO,
                          iSR_Drive_Param := "CS_MOVIKIT".CS_M2_PO,
                          oSL_Drive_Param := "CS_MOVIKIT".CS_M1_PI,
                          oSR_Drive_Param := "CS_MOVIKIT".CS_M2_PI);
END_REGION

REGION Network 2 (SCL)

   // Logika timera — włącza się tylko gdy trwa centrowanie
   #tCenteringTimer(
                   IN := "HMI_Central_Shifter".CS_Pallet_Centering,
                   PT := T#5S
   );


   IF #tCenteringTimer.Q THEN
       "HMI_Central_Shifter".CS_Pallet_Centering := FALSE;
   END_IF;

   // --- Dotychczasowa logika sterowania ---
   IF "HMI_Central_Shifter".CS_Pallet_Centering AND "iCS_SensorHoming_Left" AND NOT "iCS_SensorHoming_Right" THEN
       "HMI_Central_Shifter".CS_Pallet_Left_Move := 0;
       "HMI_Central_Shifter".CS_Pallet_Right_Move := 1;

   ELSIF "HMI_Central_Shifter".CS_Pallet_Centering AND "iCS_SensorHoming_Right" AND NOT "iCS_SensorHoming_Left" THEN
       "HMI_Central_Shifter".CS_Pallet_Left_Move := 1;
       "HMI_Central_Shifter".CS_Pallet_Right_Move := 0;

   ELSIF "HMI_Central_Shifter".CS_Pallet_Centering THEN
       "HMI_Central_Shifter".CS_Pallet_Left_Move := 0;
       "HMI_Central_Shifter".CS_Pallet_Right_Move := 0;
       "HMI_Central_Shifter".CS_Pallet_Centering := 0;
   END_IF;

   IF NOT "HMI_Central_Shifter".CS_Pallet_Centering AND #prevCentering THEN
       // Jednorazowe wyłączenie jazdy w lewo i prawo
       "HMI_Central_Shifter".CS_Pallet_Left_Move := 0;
       "HMI_Central_Shifter".CS_Pallet_Right_Move := 0;
   END_IF;

   // Aktualizacja stanu poprzedniego
   #prevCentering := "HMI_Central_Shifter".CS_Pallet_Centering;
END_REGION
END_FUNCTION_BLOCK

FUNCTION_BLOCK "Central_Auto_Control"   // FB21, LAD
{ S7_Optimized_Access := 'TRUE' }
// stored: MemoryReserve 100, SetENOAutomatically false
   VAR
      Auto_Turn_On : Bool;
      "Step" : Int;
      CS_Drive : Bool;
      SS_Go_H3 : Bool;
      SS_Go_H5 : Bool;
      SS_Go_CS : Bool;
      CS_Auto_Hyd_Up : Bool;
      CS_Auto_Hyd_Down : Bool;
      Step_Delay { S7_SetPoint := 'True'} : TON_TIME;
      Timer_active { S7_SetPoint := 'True'} : Bool;
   END_VAR
BEGIN

REGION Network 1
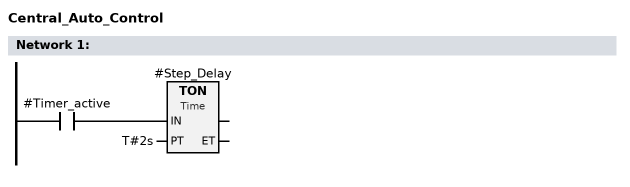
   RUNG wire#powerrail
      Contact( #Timer_active )
      { S7_Templates := "time_type := Time" } #Step_Delay.TON(pt := T#2s, et =>)
   END_RUNG
   // the same network as SCL:
   #Step_Delay(IN := #Timer_active, PT := T#2s);   // TON
END_REGION

REGION Network 2 (SCL)
   IF #Auto_Turn_On  AND "HMI_Central_Shifter".CS_Auto_Pos_Start <> 0  AND "HMI_Central_Shifter".CS_Auto_Pos_End <> 0  THEN
       IF #Step = 0 THEN  //drive CS to Start pos
           IF "CentralShifter_DB".CentralShifter_SideShifters_Instance.Hyd_Down_Status = 2 AND "CentralShifter_DB".CentralShifter_SideShifters_Instance.qLeftSide_in_Mid AND "CentralShifter_DB".CentralShifter_SideShifters_Instance.qRightSide_in_Mid AND NOT "iCS_SensorHoming_Left" AND NOT "iCS_SensorHoming_Right" THEN
               "HMI_Central_Shifter".CS_Destination_Pos := ("HMI_Central_Shifter".CS_Auto_Pos_Start MOD 10) + 6;
               #CS_Drive := 1;
           END_IF;
           IF "CentralShifter_DB".Arrived_Pos = ("HMI_Central_Shifter".CS_Auto_Pos_Start MOD 10) + 6 THEN
               #Timer_active := 1;
               IF #Step_Delay.Q THEN
                   #Step := 1;
                   #Timer_active := 0;
               END_IF;
           END_IF;

       ELSIF #Step = 1 THEN  //Drive SS to Start pos
           IF "CentralShifter_DB".Arrived_Pos <> ("HMI_Central_Shifter".CS_Auto_Pos_Start MOD 10) + 6 THEN
               #Timer_active := 1;
               IF #Step_Delay.Q THEN
                   #Step := 0;
                   #Timer_active := 0;
               END_IF;

           ELSIF "CentralShifter_DB".Arrived_Pos = ("HMI_Central_Shifter".CS_Auto_Pos_Start MOD 10) + 6 AND "CentralShifter_DB".CentralShifter_SideShifters_Instance.Hyd_Down_Status = 2 THEN
               IF "HMI_Central_Shifter".CS_Auto_Pos_Start < 10 THEN
                   #SS_Go_H5 := 1;
                   IF "CentralShifter_DB".CentralShifter_SideShifters_Instance.Sides_In_H5_Pos THEN
                       #Timer_active := 1;
                       IF #Step_Delay.Q THEN
                           #SS_Go_H5 := 0;
                           #Step := 2;
                           #Timer_active := 0;
                       END_IF;
                   END_IF;

               ELSIF "HMI_Central_Shifter".CS_Auto_Pos_Start > 10 THEN
                   #SS_Go_H3 := 1;
                   IF "CentralShifter_DB".CentralShifter_SideShifters_Instance.Sides_In_H3_Pos THEN
                       #Timer_active := 1;
                       IF #Step_Delay.Q THEN
                           #SS_Go_H3 := 0;
                           #Step := 2;
                           #Timer_active := 0;
                       END_IF;
                   END_IF;
               END_IF;
           END_IF;

       ELSIF #Step = 2 THEN  //Hyd UP SS on station
           IF NOT "CentralShifter_DB".CentralShifter_SideShifters_Instance.Sides_In_H3_Pos AND NOT "CentralShifter_DB".CentralShifter_SideShifters_Instance.Sides_In_H5_Pos AND "CentralShifter_DB".CentralShifter_SideShifters_Instance.Hyd_Down_Status = 2 THEN
               #Timer_active := 1;
               IF #Step_Delay.Q THEN
                   #Step := 1;
                   #Timer_active := 0;
               END_IF;
           ELSE
               #CS_Auto_Hyd_Up := 1;
           END_IF;
           IF "CentralShifter_DB".CentralShifter_SideShifters_Instance.Hyd_Up_Status = 2 THEN
               #CS_Auto_Hyd_Up := 0;
               #Timer_active := 1;
               IF #Step_Delay.Q THEN
                   #Step := 3;
                   #Timer_active := 0;
               END_IF;
           END_IF;

       ELSIF #Step = 3 THEN  //Drive SS to CS
           IF "CentralShifter_DB".CentralShifter_SideShifters_Instance.Hyd_Up_Status = 2 THEN
               #SS_Go_CS := 1;
               //ELSE
               //#Step := 2;
           END_IF;

           IF "CentralShifter_DB".CentralShifter_SideShifters_Instance.Sides_In_CS_Pos THEN
               #Timer_active := 1;
               IF #Step_Delay.Q THEN
                   #Step := 4;
                   #SS_Go_CS := 0;
                   #Timer_active := 0;
               END_IF;
           END_IF;

       ELSIF #Step = 4 THEN //hyd down on CS
           IF "CentralShifter_DB".CentralShifter_SideShifters_Instance.Sides_In_CS_Pos THEN
               #CS_Auto_Hyd_Down := 1;

               IF "CentralShifter_DB".CentralShifter_SideShifters_Instance.Hyd_Down_Status = 2 THEN
                   #Timer_active := 1;
                   IF #Step_Delay.Q THEN
                       #Step := 5;
                       #SS_Go_CS := 0;
                       #Timer_active := 0;
                   END_IF;
               END_IF;

           ELSE
               #SS_Go_CS := 1;
           END_IF;


       ELSIF #Step = 5 THEN //CS Drive 
           IF "CentralShifter_DB".CentralShifter_SideShifters_Instance.Hyd_Down_Status = 2 THEN
               "HMI_Central_Shifter".CS_Destination_Pos := ("HMI_Central_Shifter".CS_Auto_Pos_End MOD 10) + 6;
               #CS_Drive := 1;
           ELSE
               #Timer_active := 1;
               IF #Step_Delay.Q THEN
                   #Step := 4;
                   #Timer_active := 0;
               END_IF;
           END_IF;

           IF "CentralShifter_DB".Arrived_Pos = ("HMI_Central_Shifter".CS_Auto_Pos_End MOD 10) + 6 THEN
               #Timer_active := 1;
               IF #Step_Delay.Q THEN
                   #Step := 6;
                   #Timer_active := 0;
               END_IF;
           END_IF;

       ELSIF #Step = 6 THEN //Hyd Up on CS
           IF "CentralShifter_DB".CentralShifter_SideShifters_Instance.Sides_In_CS_Pos AND "CentralShifter_DB".Arrived_Pos = ("HMI_Central_Shifter".CS_Auto_Pos_End MOD 10) + 6 THEN
               #CS_Auto_Hyd_Up := 1;
               #SS_Go_CS := 0;
           ELSE
               #SS_Go_CS := 1;
           END_IF;
           IF "CentralShifter_DB".CentralShifter_SideShifters_Instance.Hyd_Up_Status = 2 THEN
               #Timer_active := 1;
               IF #Step_Delay.Q THEN
                   #CS_Auto_Hyd_Up := 0;
                   #SS_Go_CS := 0;
                   #Step := 7;
                   #Timer_active := 0;
               END_IF;
           END_IF;

       ELSIF #Step = 7 THEN //SS Drive to end pos
           IF "CentralShifter_DB".Arrived_Pos <> ("HMI_Central_Shifter".CS_Auto_Pos_End MOD 10) + 6 THEN
               #Timer_active := 1;
               IF #Step_Delay.Q THEN
                   #Step := 6;
                   #Timer_active := 0;
               END_IF;

           ELSIF "CentralShifter_DB".Arrived_Pos = ("HMI_Central_Shifter".CS_Auto_Pos_End MOD 10) + 6 THEN
               IF "HMI_Central_Shifter".CS_Auto_Pos_End < 10 THEN
                   #SS_Go_H5 := 1;
                   IF "CentralShifter_DB".CentralShifter_SideShifters_Instance.Sides_In_H5_Pos THEN
                       #Timer_active := 1;
                       IF #Step_Delay.Q THEN
                           #SS_Go_H5 := 0;
                           #Step := 8;
                           #Timer_active := 0;
                       END_IF;
                   END_IF;

               ELSIF "HMI_Central_Shifter".CS_Auto_Pos_End > 10 THEN
                   #SS_Go_H3 := 1;
                   IF "CentralShifter_DB".CentralShifter_SideShifters_Instance.Sides_In_H3_Pos THEN
                       #Timer_active := 1;
                       IF #Step_Delay.Q THEN
                           #SS_Go_H3 := 0;
                           #Step := 8;
                           #Timer_active := 0;
                       END_IF;
                   END_IF;
               END_IF;
           END_IF;

       ELSIF #Step = 8 THEN //Hyd down
           IF NOT "CentralShifter_DB".CentralShifter_SideShifters_Instance.Sides_In_H3_Pos AND NOT "CentralShifter_DB".CentralShifter_SideShifters_Instance.Sides_In_H5_Pos AND "CentralShifter_DB".CentralShifter_SideShifters_Instance.Hyd_Up_Status = 2 THEN
               #Timer_active := 1;
               IF #Step_Delay.Q THEN
                   #Step := 7;
                   #Timer_active := 0;
               END_IF;
           ELSE
               #CS_Auto_Hyd_Down := 1;
           END_IF;
           IF "CentralShifter_DB".CentralShifter_SideShifters_Instance.Hyd_Down_Status = 2 THEN
               #Timer_active := 1;
               IF #Step_Delay.Q THEN
                   #CS_Auto_Hyd_Down := 0;
                   #Step := 9;
                   #Timer_active := 0;
               END_IF;
           END_IF;

       ELSIF #Step = 9 THEN
           IF "CentralShifter_DB".CentralShifter_SideShifters_Instance.Hyd_Down_Status = 2 THEN
               #SS_Go_CS := 1;
           ELSE
               #Timer_active := 1;
               IF #Step_Delay.Q THEN
                   #Step := 8;
                   #Timer_active := 0;
               END_IF;
           END_IF;

           IF "CentralShifter_DB".CentralShifter_SideShifters_Instance.Sides_In_CS_Pos THEN
               #Timer_active := 1;
               IF #Step_Delay.Q THEN
                   #Step := 10;
                   #Timer_active := 0;
               END_IF;
           END_IF;
       END_IF;

   ELSE
       #CS_Drive := 0;
       #SS_Go_CS := 0;
       #SS_Go_H3 := 0;
       #SS_Go_H5 := 0;
       #CS_Auto_Hyd_Down := 0;
       #CS_Auto_Hyd_Up := 0;
       #Timer_active := 0;
       IF #Step = 10 THEN
           #Step := 0;
       END_IF;
   END_IF;
END_REGION
END_FUNCTION_BLOCK

FUNCTION_BLOCK "TorqueFB_TEL750"
{ S7_Optimized_Access := 'TRUE' }
VERSION : 0.1
   VAR_INPUT 
      enable : Bool;
      refTorque : Real;
      addTorque : Real;
      upperLimit : Real := 0.0;
      lowerLimit : Real := 0.0;
      HWIDSTW : HW_IO;   // Hardware Identifer set point slot
      HWIDZSW : HW_IO;   // Hardware Identifer actual value slot
   END_VAR

   VAR_OUTPUT 
      busy : Bool;
      inUpperLimit : Bool;
      inLowerLimit : Bool;
      actTorque : Real;
      error : Bool;
      errorID : Word;
      diaID : Word;
   END_VAR

   VAR 
      swSend : Array[0..2] of Word;
      swReceive : Word;
      sxSend : Struct
         M_ADD1 : Word;
         M_LIMIT_POS : Word;
         M_LIMIT_NEG : Word;
      END_STRUCT;
      sxReceive : Struct
         M_ACT : Word;
      END_STRUCT;
   END_VAR

   VAR_TEMP 
      piRetSFC : Int;
   END_VAR


BEGIN
	//***********************************************************************************
	//SIEMENS AG
	//(c)Copyright 2023 All Rights Reserved
	//-----------------------------------------------------------------------------
	// Library: DriveLib
	// Tested with: -
	// Engineering: TIA Portal V18
	// Restrictions: -
	// Requirements: S7-1200 / S7-1500
	// Version:    V1.0
	// Functionality: cyclic communication between a SINAMICS and a PLC via TEL750.
	//                The parametrisation of these words is described in the manual of the
	//                SINAMICS
	// Contactor: mc_gmc_mp_asia.cn@siemens.com
	//***********************************************************************************
	
	#busy := FALSE;
	#error := FALSE;
	#inUpperLimit := FALSE;
	#inLowerLimit := FALSE;
	#actTorque := 0.0;
	#errorID := 16#0000;
	#diaID := 16#0000;
	
	IF NOT #enable THEN
	    #sxSend.M_ADD1 := 16#0;
	    #sxSend.M_LIMIT_POS := 16#4000;
	    #sxSend.M_LIMIT_NEG := 16#C000;
	END_IF;
	
	IF #enable THEN
	    IF #refTorque <= 0.0 THEN
	        #error := TRUE;
	        #errorID := 16#8001;
	    ELSIF #upperLimit > #refTorque THEN
	        #error := TRUE;
	        #errorID := 16#8002;
	    ELSIF #lowerLimit < - #refTorque THEN
	        #error := TRUE;
	        #errorID := 16#8003;
	    ELSIF #upperLimit<=#lowerLimit THEN
	        #error := TRUE;
	        #errorID := 16#8004;
	    ELSIF #upperLimit<0.0 THEN
	        #error := TRUE;
	        #errorID := 16#8005;
	    ELSIF #lowerLimit>0.0 THEN
	        #error := TRUE;
	        #errorID := 16#8006;
	    ELSE
	        #error := FALSE;
	        #errorID := 16#0000;
	    END_IF;
	    
	    IF NOT #error THEN
	        #busy := TRUE;
	        #sxSend.M_ADD1 := INT_TO_WORD(REAL_TO_INT(#addTorque * 16384.0 / #refTorque));
	        #sxSend.M_LIMIT_POS := INT_TO_WORD(REAL_TO_INT(#upperLimit * 16384.0 / #refTorque));
	        #sxSend.M_LIMIT_NEG := INT_TO_WORD(REAL_TO_INT(#lowerLimit * 16384.0 / #refTorque));
	    ELSE
	        #busy := FALSE;
	        #sxSend.M_ADD1 := 16#0;
	        #sxSend.M_LIMIT_POS := 16#4000;
	        #sxSend.M_LIMIT_NEG := 16#C000;
	    END_IF;
	END_IF;
	#swSend[0] := #sxSend.M_ADD1;
	#swSend[1] := #sxSend.M_LIMIT_POS;
	#swSend[2] := #sxSend.M_LIMIT_NEG;
	
	#piRetSFC := DPWR_DAT(LADDR := #HWIDSTW,
	                      RECORD := #swSend);
	#diaID := INT_TO_WORD(#piRetSFC);
	
	IF #piRetSFC = 0 THEN
	    #piRetSFC := DPRD_DAT(LADDR := #HWIDZSW, RECORD => #swReceive);
	    #diaID := INT_TO_WORD(#piRetSFC);
	    IF #piRetSFC = 0 THEN
	        #sxReceive.M_ACT := #swReceive;
	    ELSE
	        #error := TRUE;
	        #errorID := 16#8008;
	        #sxReceive.M_ACT := 16#000;
	    END_IF;
	ELSE
	    #error := TRUE;
	    #errorID := 16#8007;
	END_IF;
	
	#actTorque := INT_TO_REAL(WORD_TO_INT(#sxReceive.M_ACT)) * #refTorque / 16384.0;
	
	IF #enable THEN
	    
	    IF #upperLimit > 0.0 THEN
	        IF #actTorque >= #upperLimit THEN
	            #inUpperLimit := TRUE;
	        END_IF;
	    ELSE
	        IF #actTorque >= #refTorque THEN
	            #inUpperLimit := TRUE;
	        END_IF;
	    END_IF;
	    IF #lowerLimit < 0.0 THEN
	        IF #actTorque <= #lowerLimit THEN
	            #inLowerLimit := TRUE;
	        END_IF;
	    ELSE
	        IF #actTorque <= -#refTorque THEN
	            #inLowerLimit := TRUE;
	        END_IF;
	    END_IF;
	END_IF;
	        
END_FUNCTION_BLOCK

FUNCTION "Lights" : Void   // FC6, LAD
{ S7_Optimized_Access := 'TRUE' }
// stored: SetENOAutomatically false
   VAR_TEMP
      Column_13_14_CS : Bool;
      Column_14_08_CS : Bool;
      i : SInt;
      Hmi_Button_Drive : Bool;
   END_VAR
BEGIN

REGION Network 1: Safety
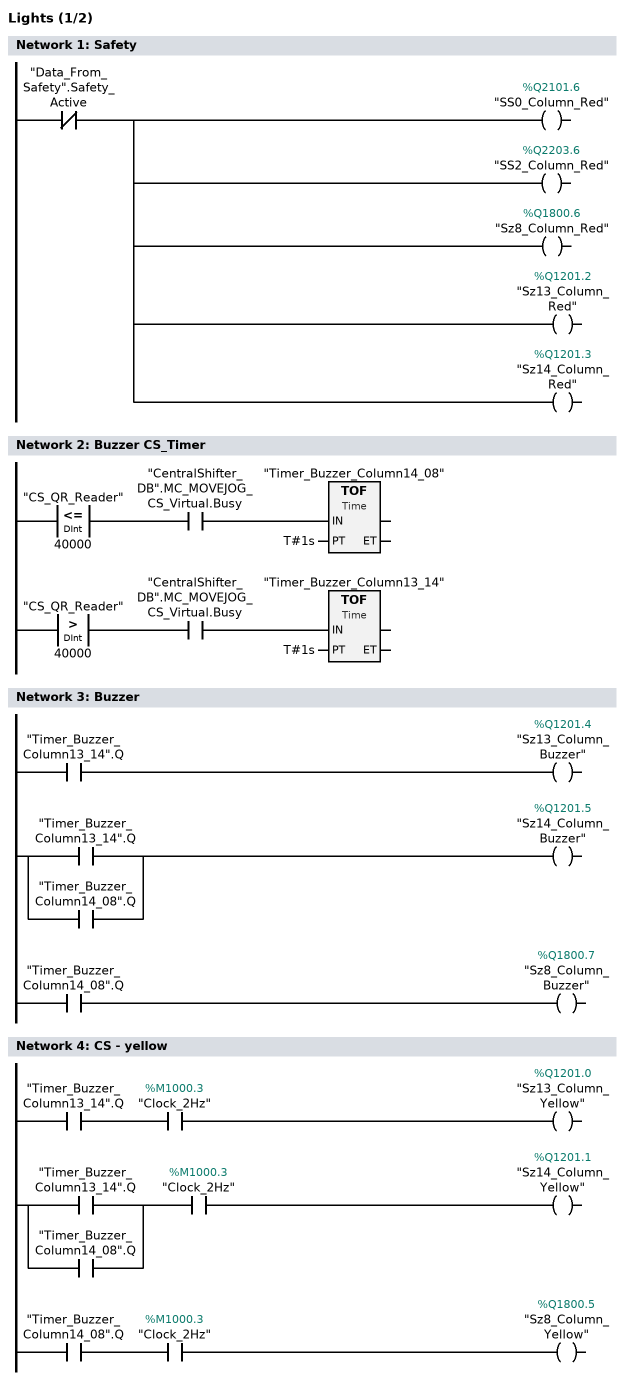
   RUNG wire#powerrail
      I_Contact( "Data_From_Safety".Safety_Active )
      wire#w1
      Coil( "SS0_Column_Red" )
   END_RUNG
   RUNG wire#w1
      Coil( "SS2_Column_Red" )
   END_RUNG
   RUNG wire#w1
      Coil( "Sz8_Column_Red" )
   END_RUNG
   RUNG wire#w1
      Coil( "Sz13_Column_Red" )
   END_RUNG
   RUNG wire#w1
      Coil( "Sz14_Column_Red" )
   END_RUNG
   // the same network as SCL:
   "SS0_Column_Red" := NOT "Data_From_Safety".Safety_Active;
   "SS2_Column_Red" := NOT "Data_From_Safety".Safety_Active;
   "Sz8_Column_Red" := NOT "Data_From_Safety".Safety_Active;
   "Sz13_Column_Red" := NOT "Data_From_Safety".Safety_Active;
   "Sz14_Column_Red" := NOT "Data_From_Safety".Safety_Active;
END_REGION

REGION Network 2: Buzzer CS_Timer
   RUNG wire#powerrail
      { S7_Templates := "SrcType := DInt" } LE_Contact(in1 := "CS_QR_Reader", in2 := 40000)
      Contact( "CentralShifter_DB".MC_MOVEJOG_CS_Virtual.Busy )
      { S7_Templates := "time_type := Time" } "Timer_Buzzer_Column14_08".TOF(pt := T#1s, et =>)
   END_RUNG
   RUNG wire#powerrail
      { S7_Templates := "SrcType := DInt" } GT_Contact(in1 := "CS_QR_Reader", in2 := 40000)
      Contact( "CentralShifter_DB".MC_MOVEJOG_CS_Virtual.Busy )
      { S7_Templates := "time_type := Time" } "Timer_Buzzer_Column13_14".TOF(pt := T#1s, et =>)
   END_RUNG
   // the same network as SCL:
   "Timer_Buzzer_Column14_08".TOF(IN := ("CS_QR_Reader" <= 40000) AND "CentralShifter_DB".MC_MOVEJOG_CS_Virtual.Busy,
                           PT := T#1s);
   "Timer_Buzzer_Column13_14".TOF(IN := ("CS_QR_Reader" > 40000) AND "CentralShifter_DB".MC_MOVEJOG_CS_Virtual.Busy,
                           PT := T#1s);
END_REGION

REGION Network 3: Buzzer
   RUNG wire#powerrail
      Contact( "Timer_Buzzer_Column13_14".Q )
      Coil( "Sz13_Column_Buzzer" )
   END_RUNG
   RUNG wire#powerrail
      Contact( "Timer_Buzzer_Column13_14".Q )
      wire#w1
      Coil( "Sz14_Column_Buzzer" )
   END_RUNG
   RUNG wire#powerrail
      Contact( "Timer_Buzzer_Column14_08".Q )
   END_RUNG wire#w1
   RUNG wire#powerrail
      Contact( "Timer_Buzzer_Column14_08".Q )
      Coil( "Sz8_Column_Buzzer" )
   END_RUNG
   // the same network as SCL:
   "Sz13_Column_Buzzer" := "Timer_Buzzer_Column13_14".Q;
   "Sz14_Column_Buzzer" := "Timer_Buzzer_Column13_14".Q OR "Timer_Buzzer_Column14_08".Q;
   "Sz8_Column_Buzzer" := "Timer_Buzzer_Column14_08".Q;
END_REGION

REGION Network 4: CS - yellow
   RUNG wire#powerrail
      Contact( "Timer_Buzzer_Column13_14".Q )
      Contact( "Clock_2Hz" )
      Coil( "Sz13_Column_Yellow" )
   END_RUNG
   RUNG wire#powerrail
      Contact( "Timer_Buzzer_Column13_14".Q )
      wire#w1
      Contact( "Clock_2Hz" )
      Coil( "Sz14_Column_Yellow" )
   END_RUNG
   RUNG wire#powerrail
      Contact( "Timer_Buzzer_Column14_08".Q )
   END_RUNG wire#w1
   RUNG wire#powerrail
      Contact( "Timer_Buzzer_Column14_08".Q )
      Contact( "Clock_2Hz" )
      Coil( "Sz8_Column_Yellow" )
   END_RUNG
   // the same network as SCL:
   "Sz13_Column_Yellow" := "Timer_Buzzer_Column13_14".Q AND "Clock_2Hz";
   "Sz14_Column_Yellow" := ("Timer_Buzzer_Column13_14".Q OR "Timer_Buzzer_Column14_08".Q) AND "Clock_2Hz";
   "Sz8_Column_Yellow" := "Timer_Buzzer_Column14_08".Q AND "Clock_2Hz";
END_REGION

REGION Network 5: Safety barriers SS1
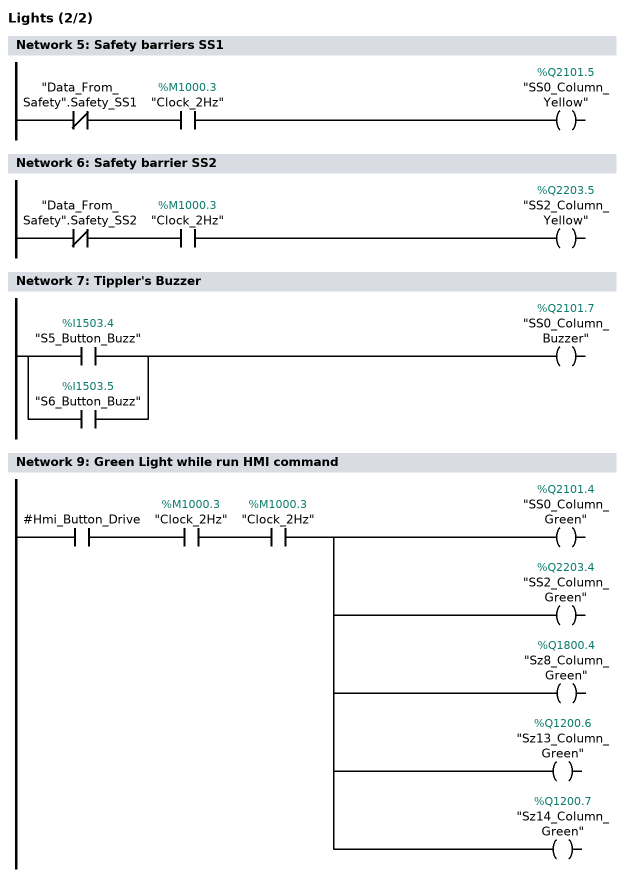
   RUNG wire#powerrail
      I_Contact( "Data_From_Safety".Safety_SS1 )
      Contact( "Clock_2Hz" )
      Coil( "SS0_Column_Yellow" )
   END_RUNG
   // the same network as SCL:
   "SS0_Column_Yellow" := NOT "Data_From_Safety".Safety_SS1 AND "Clock_2Hz";
END_REGION

REGION Network 6: Safety barrier SS2
   RUNG wire#powerrail
      I_Contact( "Data_From_Safety".Safety_SS2 )
      Contact( "Clock_2Hz" )
      Coil( "SS2_Column_Yellow" )
   END_RUNG
   // the same network as SCL:
   "SS2_Column_Yellow" := NOT "Data_From_Safety".Safety_SS2 AND "Clock_2Hz";
END_REGION

REGION Network 7: Tippler's Buzzer
   RUNG wire#powerrail
      Contact( "S5_Button_Buzz" )
      wire#w1
      Coil( "SS0_Column_Buzzer" )
   END_RUNG
   RUNG wire#powerrail
      Contact( "S6_Button_Buzz" )
   END_RUNG wire#w1
   // the same network as SCL:
   "SS0_Column_Buzzer" := "S5_Button_Buzz" OR "S6_Button_Buzz";
END_REGION

REGION Network 8 (SCL): Any run button from HMI
       FOR #i := 1 TO 12 DO
           #Hmi_Button_Drive :=
           "HMI_Pallets".Run_Command_left_ROW1[#i] OR
           "HMI_Pallets".Run_Command_left_ROW2[#i] OR
           "HMI_Pallets".Run_Command_left_ROW4[#i] OR
           "HMI_Pallets".Run_Command_right_ROW1[#i] OR
           "HMI_Pallets".Run_Command_right_ROW2[#i] OR
           "HMI_Pallets".Run_Command_right_ROW4[#i];
       END_FOR;
END_REGION

REGION Network 9: Green Light while run HMI command
   RUNG wire#powerrail
      Contact( #Hmi_Button_Drive )
      Contact( "Clock_2Hz" )
      Contact( "Clock_2Hz" )
      wire#w1
      Coil( "SS0_Column_Green" )
   END_RUNG
   RUNG wire#w1
      Coil( "SS2_Column_Green" )
   END_RUNG
   RUNG wire#w1
      Coil( "Sz8_Column_Green" )
   END_RUNG
   RUNG wire#w1
      Coil( "Sz13_Column_Green" )
   END_RUNG
   RUNG wire#w1
      Coil( "Sz14_Column_Green" )
   END_RUNG
   // the same network as SCL:
   "SS0_Column_Green" := #Hmi_Button_Drive AND "Clock_2Hz" AND "Clock_2Hz";
   "SS2_Column_Green" := "SS0_Column_Green";
   "Sz8_Column_Green" := "SS0_Column_Green";
   "Sz13_Column_Green" := "SS0_Column_Green";
   "Sz14_Column_Green" := "SS0_Column_Green";
END_REGION
END_FUNCTION

FUNCTION_BLOCK "CC_Main"   // FB100, LAD
{ S7_Optimized_Access := 'TRUE' }
// stored: AutoNumber false, MemoryReserve 100, SetENOAutomatically false
   VAR_INPUT
      HMI_Reset : Bool;
      ST23_Selected : Bool;
      CNT_DownPos1 : Bool;
      CNT_DownPos2 : Bool;
      CNT_UpPos1 : Bool;
      CNT_UpPos2 : Bool;
      Hydraulic_Roller_DownPos1 : Bool;
      Hydraulic_Roller_DownPos2 : Bool;
      Hydraulic_Roller_UpPos1 : Bool;
      Hydraulic_Roller_UpPos2 : Bool;
      Drive_Roller_DownPos1 : Bool;
      Drive_Roller_DownPos2 : Bool;
      Drive_Roller_UpPos1 : Bool;
      Drive_Roller_UpPos2 : Bool;
      Module_DownPos1 : Bool;
      Module_DownPos2 : Bool;
      Module_UpPos1 : Bool;
      Module_UpPos2 : Bool;
   END_VAR
   VAR_OUTPUT
      Hydraulic_Main_Valve_Control : Bool;
   END_VAR
   VAR
      Hydraulic_Unit_Active : Bool;
      Any_Valve_Active : Bool;
      HydUnitTimerOff { S7_SetPoint := 'True'} : TON_TIME;
      HydraulicUnit_MC_Power { S7_SetPoint := 'True'} : MC_POWER;
      HydraulicUnit_MC_MoveJog { S7_SetPoint := 'True'} : MC_MOVEJOG;
      HydraulicUnit_MC_Reset { S7_SetPoint := 'True'} : MC_RESET;
      Vibrator_Control_MOD1 { S7_SetPoint := 'True'} : "CC_Vibrator_Control";
      Vibrator_Control_MOD2 { S7_SetPoint := 'True'} : "CC_Vibrator_Control";
      Vibrator_Control_MOD3 { S7_SetPoint := 'True'} : "CC_Vibrator_Control";
      Module_Control_ST23 { S7_SetPoint := 'True'} : "CC_Vib_Modules";
      ST23_UP_whenMoving { S7_SetPoint := 'True'} : Bool;
      ST24_UP_whenMoving : Bool;
      ST25_UP_whenMoving : Bool;
      MC_Power_Vib1 { S7_SetPoint := 'True'} : MC_POWER;
      MC_RESET_Vib1 { S7_SetPoint := 'True'} : MC_RESET;
      MC_MOVEJOG_Vib1 { S7_SetPoint := 'True'} : MC_MOVEJOG;
      ST24_DriveRollsUP { S7_SetPoint := 'True'} : Bool;
      ST24_DriveRollsDown : Bool;
      ST25_DriveRollsUp : Bool;
      ST25_DriveRollsDown : Bool;
      ST23_Station_Control { S7_SetPoint := 'True'} : "CC_Station_Control";
      ST24_Station_Control { S7_SetPoint := 'True'} : "CC_Station_Control";
      ST25_Station_Control { S7_SetPoint := 'True'} : "CC_Station_Control";
      ST24_Selected : Bool;
   END_VAR
   VAR CONSTANT
      STEP_RETRACT : Int := 1;
      STEP_MOVING : Int := 2;
      STEP_EXTEND : Int := 3;
   END_VAR
BEGIN

REGION Network 1
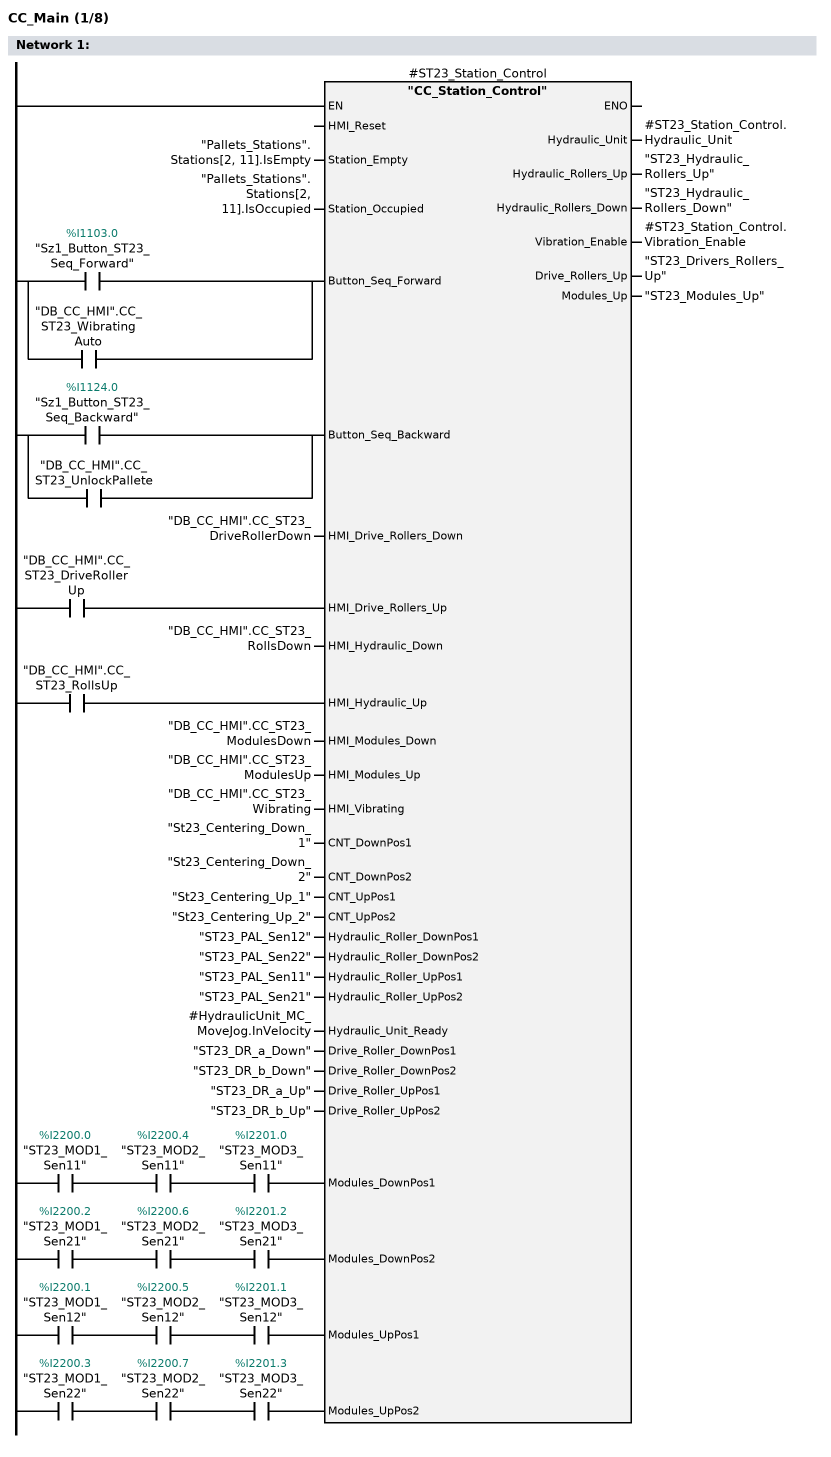
   RUNG wire#powerrail
      #ST23_Station_Control(Button_Seq_Forward := wire#w1, Button_Seq_Backward := wire#w2, HMI_Drive_Rollers_Up := wire#w3, HMI_Hydraulic_Up := wire#w4, Modules_DownPos1 := wire#w5, Modules_DownPos2 := wire#w6, Modules_UpPos1 := wire#w7, Modules_UpPos2 := wire#w8, HMI_Reset :=, Station_Empty := "Pallets_Stations".Stations[2, 11].IsEmpty, Station_Occupied := "Pallets_Stations".Stations[2, 11].IsOccupied, HMI_Drive_Rollers_Down := "DB_CC_HMI".CC_ST23_DriveRollerDown, HMI_Hydraulic_Down := "DB_CC_HMI".CC_ST23_RollsDown, HMI_Modules_Down := "DB_CC_HMI".CC_ST23_ModulesDown, HMI_Modules_Up := "DB_CC_HMI".CC_ST23_ModulesUp, HMI_Vibrating := "DB_CC_HMI".CC_ST23_Wibrating, CNT_DownPos1 := "St23_Centering_Down_1", CNT_DownPos2 := "St23_Centering_Down_2", CNT_UpPos1 := "St23_Centering_Up_1", CNT_UpPos2 := "St23_Centering_Up_2", Hydraulic_Roller_DownPos1 := "ST23_PAL_Sen12", Hydraulic_Roller_DownPos2 := "ST23_PAL_Sen22", Hydraulic_Roller_UpPos1 := "ST23_PAL_Sen11", Hydraulic_Roller_UpPos2 := "ST23_PAL_Sen21", Hydraulic_Unit_Ready := #HydraulicUnit_MC_MoveJog.InVelocity, Drive_Roller_DownPos1 := "ST23_DR_a_Down", Drive_Roller_DownPos2 := "ST23_DR_b_Down", Drive_Roller_UpPos1 := "ST23_DR_a_Up", Drive_Roller_UpPos2 := "ST23_DR_b_Up", Hydraulic_Unit => #ST23_Station_Control.Hydraulic_Unit, Hydraulic_Rollers_Up => "ST23_Hydraulic_Rollers_Up", Hydraulic_Rollers_Down => "ST23_Hydraulic_Rollers_Down", Vibration_Enable => #ST23_Station_Control.Vibration_Enable, Drive_Rollers_Up => "ST23_Drivers_Rollers_Up", Modules_Up => "ST23_Modules_Up")
   END_RUNG
   RUNG wire#powerrail
      Contact( "Sz1_Button_ST23_Seq_Forward" )
   END_RUNG wire#w1
   RUNG wire#powerrail
      Contact( "DB_CC_HMI".CC_ST23_WibratingAuto )
   END_RUNG wire#w1
   RUNG wire#powerrail
      Contact( "Sz1_Button_ST23_Seq_Backward" )
   END_RUNG wire#w2
   RUNG wire#powerrail
      Contact( "DB_CC_HMI".CC_ST23_UnlockPallete )
   END_RUNG wire#w2
   RUNG wire#powerrail
      Contact( "DB_CC_HMI".CC_ST23_DriveRollerUp )
   END_RUNG wire#w3
   RUNG wire#powerrail
      Contact( "DB_CC_HMI".CC_ST23_RollsUp )
   END_RUNG wire#w4
   RUNG wire#powerrail
      Contact( "ST23_MOD1_Sen11" )
      Contact( "ST23_MOD2_Sen11" )
      Contact( "ST23_MOD3_Sen11" )
   END_RUNG wire#w5
   RUNG wire#powerrail
      Contact( "ST23_MOD1_Sen21" )
      Contact( "ST23_MOD2_Sen21" )
      Contact( "ST23_MOD3_Sen21" )
   END_RUNG wire#w6
   RUNG wire#powerrail
      Contact( "ST23_MOD1_Sen12" )
      Contact( "ST23_MOD2_Sen12" )
      Contact( "ST23_MOD3_Sen12" )
   END_RUNG wire#w7
   RUNG wire#powerrail
      Contact( "ST23_MOD1_Sen22" )
      Contact( "ST23_MOD2_Sen22" )
      Contact( "ST23_MOD3_Sen22" )
   END_RUNG wire#w8
   // the same network as SCL:
   #ST23_Station_Control(Station_Empty := "Pallets_Stations".Stations[2, 11].IsEmpty,   // "CC_Station_Control"
                         Station_Occupied := "Pallets_Stations".Stations[2, 11].IsOccupied,
                         Button_Seq_Forward := "Sz1_Button_ST23_Seq_Forward" OR "DB_CC_HMI".CC_ST23_WibratingAuto,
                         Button_Seq_Backward := "Sz1_Button_ST23_Seq_Backward" OR "DB_CC_HMI".CC_ST23_UnlockPallete,
                         HMI_Drive_Rollers_Down := "DB_CC_HMI".CC_ST23_DriveRollerDown,
                         HMI_Drive_Rollers_Up := "DB_CC_HMI".CC_ST23_DriveRollerUp,
                         HMI_Hydraulic_Down := "DB_CC_HMI".CC_ST23_RollsDown,
                         HMI_Hydraulic_Up := "DB_CC_HMI".CC_ST23_RollsUp,
                         HMI_Modules_Down := "DB_CC_HMI".CC_ST23_ModulesDown,
                         HMI_Modules_Up := "DB_CC_HMI".CC_ST23_ModulesUp,
                         HMI_Vibrating := "DB_CC_HMI".CC_ST23_Wibrating,
                         CNT_DownPos1 := "St23_Centering_Down_1",
                         CNT_DownPos2 := "St23_Centering_Down_2",
                         CNT_UpPos1 := "St23_Centering_Up_1",
                         CNT_UpPos2 := "St23_Centering_Up_2",
                         Hydraulic_Roller_DownPos1 := "ST23_PAL_Sen12",
                         Hydraulic_Roller_DownPos2 := "ST23_PAL_Sen22",
                         Hydraulic_Roller_UpPos1 := "ST23_PAL_Sen11",
                         Hydraulic_Roller_UpPos2 := "ST23_PAL_Sen21",
                         Hydraulic_Unit_Ready := #HydraulicUnit_MC_MoveJog.InVelocity,
                         Drive_Roller_DownPos1 := "ST23_DR_a_Down",
                         Drive_Roller_DownPos2 := "ST23_DR_b_Down",
                         Drive_Roller_UpPos1 := "ST23_DR_a_Up",
                         Drive_Roller_UpPos2 := "ST23_DR_b_Up",
                         Modules_DownPos1 := "ST23_MOD1_Sen11" AND "ST23_MOD2_Sen11" AND "ST23_MOD3_Sen11",
                         Modules_DownPos2 := "ST23_MOD1_Sen21" AND "ST23_MOD2_Sen21" AND "ST23_MOD3_Sen21",
                         Modules_UpPos1 := "ST23_MOD1_Sen12" AND "ST23_MOD2_Sen12" AND "ST23_MOD3_Sen12",
                         Modules_UpPos2 := "ST23_MOD1_Sen22" AND "ST23_MOD2_Sen22" AND "ST23_MOD3_Sen22",
                         Hydraulic_Unit => #ST23_Station_Control.Hydraulic_Unit,
                         Hydraulic_Rollers_Up => "ST23_Hydraulic_Rollers_Up",
                         Hydraulic_Rollers_Down => "ST23_Hydraulic_Rollers_Down",
                         Vibration_Enable => #ST23_Station_Control.Vibration_Enable,
                         Drive_Rollers_Up => "ST23_Drivers_Rollers_Up",
                         Modules_Up => "ST23_Modules_Up");
END_REGION

REGION Network 2
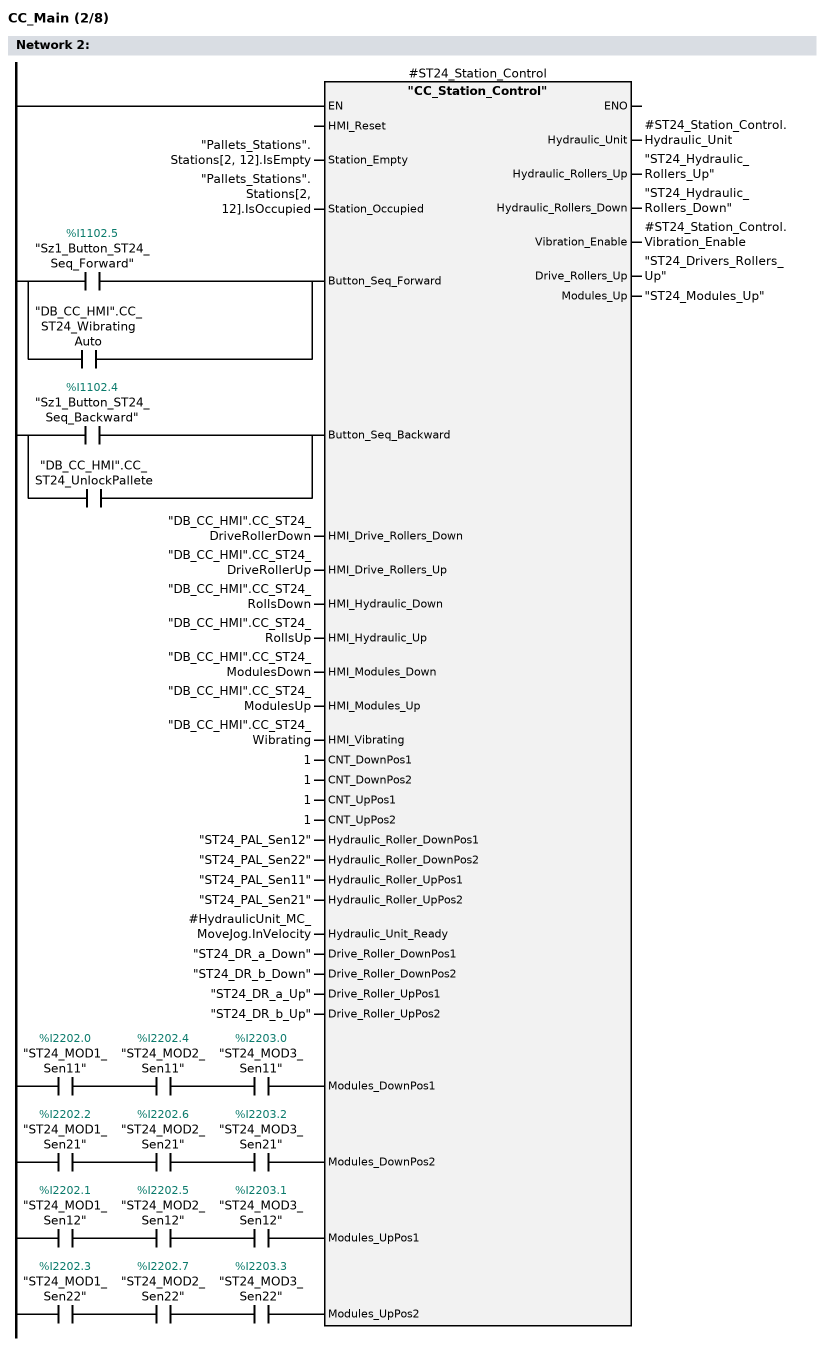
   RUNG wire#powerrail
      #ST24_Station_Control(Button_Seq_Forward := wire#w1, Button_Seq_Backward := wire#w2, Modules_DownPos1 := wire#w3, Modules_DownPos2 := wire#w4, Modules_UpPos1 := wire#w5, Modules_UpPos2 := wire#w6, HMI_Reset :=, Station_Empty := "Pallets_Stations".Stations[2, 12].IsEmpty, Station_Occupied := "Pallets_Stations".Stations[2, 12].IsOccupied, HMI_Drive_Rollers_Down := "DB_CC_HMI".CC_ST24_DriveRollerDown, HMI_Drive_Rollers_Up := "DB_CC_HMI".CC_ST24_DriveRollerUp, HMI_Hydraulic_Down := "DB_CC_HMI".CC_ST24_RollsDown, HMI_Hydraulic_Up := "DB_CC_HMI".CC_ST24_RollsUp, HMI_Modules_Down := "DB_CC_HMI".CC_ST24_ModulesDown, HMI_Modules_Up := "DB_CC_HMI".CC_ST24_ModulesUp, HMI_Vibrating := "DB_CC_HMI".CC_ST24_Wibrating, CNT_DownPos1 := 1, CNT_DownPos2 := 1, CNT_UpPos1 := 1, CNT_UpPos2 := 1, Hydraulic_Roller_DownPos1 := "ST24_PAL_Sen12", Hydraulic_Roller_DownPos2 := "ST24_PAL_Sen22", Hydraulic_Roller_UpPos1 := "ST24_PAL_Sen11", Hydraulic_Roller_UpPos2 := "ST24_PAL_Sen21", Hydraulic_Unit_Ready := #HydraulicUnit_MC_MoveJog.InVelocity, Drive_Roller_DownPos1 := "ST24_DR_a_Down", Drive_Roller_DownPos2 := "ST24_DR_b_Down", Drive_Roller_UpPos1 := "ST24_DR_a_Up", Drive_Roller_UpPos2 := "ST24_DR_b_Up", Hydraulic_Unit => #ST24_Station_Control.Hydraulic_Unit, Hydraulic_Rollers_Up => "ST24_Hydraulic_Rollers_Up", Hydraulic_Rollers_Down => "ST24_Hydraulic_Rollers_Down", Vibration_Enable => #ST24_Station_Control.Vibration_Enable, Drive_Rollers_Up => "ST24_Drivers_Rollers_Up", Modules_Up => "ST24_Modules_Up")
   END_RUNG
   RUNG wire#powerrail
      Contact( "Sz1_Button_ST24_Seq_Forward" )
   END_RUNG wire#w1
   RUNG wire#powerrail
      Contact( "DB_CC_HMI".CC_ST24_WibratingAuto )
   END_RUNG wire#w1
   RUNG wire#powerrail
      Contact( "Sz1_Button_ST24_Seq_Backward" )
   END_RUNG wire#w2
   RUNG wire#powerrail
      Contact( "DB_CC_HMI".CC_ST24_UnlockPallete )
   END_RUNG wire#w2
   RUNG wire#powerrail
      Contact( "ST24_MOD1_Sen11" )
      Contact( "ST24_MOD2_Sen11" )
      Contact( "ST24_MOD3_Sen11" )
   END_RUNG wire#w3
   RUNG wire#powerrail
      Contact( "ST24_MOD1_Sen21" )
      Contact( "ST24_MOD2_Sen21" )
      Contact( "ST24_MOD3_Sen21" )
   END_RUNG wire#w4
   RUNG wire#powerrail
      Contact( "ST24_MOD1_Sen12" )
      Contact( "ST24_MOD2_Sen12" )
      Contact( "ST24_MOD3_Sen12" )
   END_RUNG wire#w5
   RUNG wire#powerrail
      Contact( "ST24_MOD1_Sen22" )
      Contact( "ST24_MOD2_Sen22" )
      Contact( "ST24_MOD3_Sen22" )
   END_RUNG wire#w6
   // the same network as SCL:
   #ST24_Station_Control(Station_Empty := "Pallets_Stations".Stations[2, 12].IsEmpty,   // "CC_Station_Control"
                         Station_Occupied := "Pallets_Stations".Stations[2, 12].IsOccupied,
                         Button_Seq_Forward := "Sz1_Button_ST24_Seq_Forward" OR "DB_CC_HMI".CC_ST24_WibratingAuto,
                         Button_Seq_Backward := "Sz1_Button_ST24_Seq_Backward" OR "DB_CC_HMI".CC_ST24_UnlockPallete,
                         HMI_Drive_Rollers_Down := "DB_CC_HMI".CC_ST24_DriveRollerDown,
                         HMI_Drive_Rollers_Up := "DB_CC_HMI".CC_ST24_DriveRollerUp,
                         HMI_Hydraulic_Down := "DB_CC_HMI".CC_ST24_RollsDown,
                         HMI_Hydraulic_Up := "DB_CC_HMI".CC_ST24_RollsUp,
                         HMI_Modules_Down := "DB_CC_HMI".CC_ST24_ModulesDown,
                         HMI_Modules_Up := "DB_CC_HMI".CC_ST24_ModulesUp,
                         HMI_Vibrating := "DB_CC_HMI".CC_ST24_Wibrating,
                         CNT_DownPos1 := 1,
                         CNT_DownPos2 := 1,
                         CNT_UpPos1 := 1,
                         CNT_UpPos2 := 1,
                         Hydraulic_Roller_DownPos1 := "ST24_PAL_Sen12",
                         Hydraulic_Roller_DownPos2 := "ST24_PAL_Sen22",
                         Hydraulic_Roller_UpPos1 := "ST24_PAL_Sen11",
                         Hydraulic_Roller_UpPos2 := "ST24_PAL_Sen21",
                         Hydraulic_Unit_Ready := #HydraulicUnit_MC_MoveJog.InVelocity,
                         Drive_Roller_DownPos1 := "ST24_DR_a_Down",
                         Drive_Roller_DownPos2 := "ST24_DR_b_Down",
                         Drive_Roller_UpPos1 := "ST24_DR_a_Up",
                         Drive_Roller_UpPos2 := "ST24_DR_b_Up",
                         Modules_DownPos1 := "ST24_MOD1_Sen11" AND "ST24_MOD2_Sen11" AND "ST24_MOD3_Sen11",
                         Modules_DownPos2 := "ST24_MOD1_Sen21" AND "ST24_MOD2_Sen21" AND "ST24_MOD3_Sen21",
                         Modules_UpPos1 := "ST24_MOD1_Sen12" AND "ST24_MOD2_Sen12" AND "ST24_MOD3_Sen12",
                         Modules_UpPos2 := "ST24_MOD1_Sen22" AND "ST24_MOD2_Sen22" AND "ST24_MOD3_Sen22",
                         Hydraulic_Unit => #ST24_Station_Control.Hydraulic_Unit,
                         Hydraulic_Rollers_Up => "ST24_Hydraulic_Rollers_Up",
                         Hydraulic_Rollers_Down => "ST24_Hydraulic_Rollers_Down",
                         Vibration_Enable => #ST24_Station_Control.Vibration_Enable,
                         Drive_Rollers_Up => "ST24_Drivers_Rollers_Up",
                         Modules_Up => "ST24_Modules_Up");
END_REGION

REGION Network 3
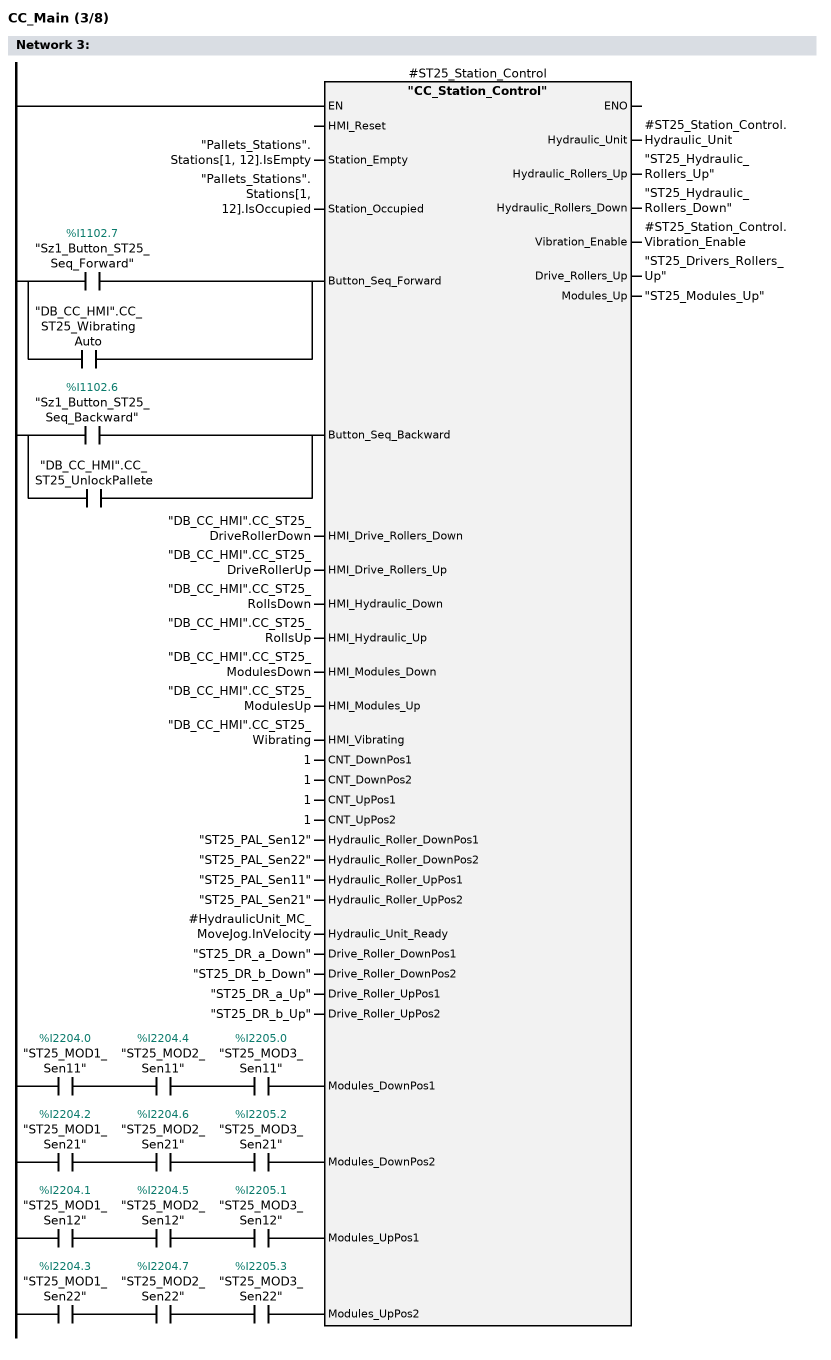
   RUNG wire#powerrail
      #ST25_Station_Control(Button_Seq_Forward := wire#w1, Button_Seq_Backward := wire#w2, Modules_DownPos1 := wire#w3, Modules_DownPos2 := wire#w4, Modules_UpPos1 := wire#w5, Modules_UpPos2 := wire#w6, HMI_Reset :=, Station_Empty := "Pallets_Stations".Stations[1, 12].IsEmpty, Station_Occupied := "Pallets_Stations".Stations[1, 12].IsOccupied, HMI_Drive_Rollers_Down := "DB_CC_HMI".CC_ST25_DriveRollerDown, HMI_Drive_Rollers_Up := "DB_CC_HMI".CC_ST25_DriveRollerUp, HMI_Hydraulic_Down := "DB_CC_HMI".CC_ST25_RollsDown, HMI_Hydraulic_Up := "DB_CC_HMI".CC_ST25_RollsUp, HMI_Modules_Down := "DB_CC_HMI".CC_ST25_ModulesDown, HMI_Modules_Up := "DB_CC_HMI".CC_ST25_ModulesUp, HMI_Vibrating := "DB_CC_HMI".CC_ST25_Wibrating, CNT_DownPos1 := 1, CNT_DownPos2 := 1, CNT_UpPos1 := 1, CNT_UpPos2 := 1, Hydraulic_Roller_DownPos1 := "ST25_PAL_Sen12", Hydraulic_Roller_DownPos2 := "ST25_PAL_Sen22", Hydraulic_Roller_UpPos1 := "ST25_PAL_Sen11", Hydraulic_Roller_UpPos2 := "ST25_PAL_Sen21", Hydraulic_Unit_Ready := #HydraulicUnit_MC_MoveJog.InVelocity, Drive_Roller_DownPos1 := "ST25_DR_a_Down", Drive_Roller_DownPos2 := "ST25_DR_b_Down", Drive_Roller_UpPos1 := "ST25_DR_a_Up", Drive_Roller_UpPos2 := "ST25_DR_b_Up", Hydraulic_Unit => #ST25_Station_Control.Hydraulic_Unit, Hydraulic_Rollers_Up => "ST25_Hydraulic_Rollers_Up", Hydraulic_Rollers_Down => "ST25_Hydraulic_Rollers_Down", Vibration_Enable => #ST25_Station_Control.Vibration_Enable, Drive_Rollers_Up => "ST25_Drivers_Rollers_Up", Modules_Up => "ST25_Modules_Up")
   END_RUNG
   RUNG wire#powerrail
      Contact( "Sz1_Button_ST25_Seq_Forward" )
   END_RUNG wire#w1
   RUNG wire#powerrail
      Contact( "DB_CC_HMI".CC_ST25_WibratingAuto )
   END_RUNG wire#w1
   RUNG wire#powerrail
      Contact( "Sz1_Button_ST25_Seq_Backward" )
   END_RUNG wire#w2
   RUNG wire#powerrail
      Contact( "DB_CC_HMI".CC_ST25_UnlockPallete )
   END_RUNG wire#w2
   RUNG wire#powerrail
      Contact( "ST25_MOD1_Sen11" )
      Contact( "ST25_MOD2_Sen11" )
      Contact( "ST25_MOD3_Sen11" )
   END_RUNG wire#w3
   RUNG wire#powerrail
      Contact( "ST25_MOD1_Sen21" )
      Contact( "ST25_MOD2_Sen21" )
      Contact( "ST25_MOD3_Sen21" )
   END_RUNG wire#w4
   RUNG wire#powerrail
      Contact( "ST25_MOD1_Sen12" )
      Contact( "ST25_MOD2_Sen12" )
      Contact( "ST25_MOD3_Sen12" )
   END_RUNG wire#w5
   RUNG wire#powerrail
      Contact( "ST25_MOD1_Sen22" )
      Contact( "ST25_MOD2_Sen22" )
      Contact( "ST25_MOD3_Sen22" )
   END_RUNG wire#w6
   // the same network as SCL:
   #ST25_Station_Control(Station_Empty := "Pallets_Stations".Stations[1, 12].IsEmpty,   // "CC_Station_Control"
                         Station_Occupied := "Pallets_Stations".Stations[1, 12].IsOccupied,
                         Button_Seq_Forward := "Sz1_Button_ST25_Seq_Forward" OR "DB_CC_HMI".CC_ST25_WibratingAuto,
                         Button_Seq_Backward := "Sz1_Button_ST25_Seq_Backward" OR "DB_CC_HMI".CC_ST25_UnlockPallete,
                         HMI_Drive_Rollers_Down := "DB_CC_HMI".CC_ST25_DriveRollerDown,
                         HMI_Drive_Rollers_Up := "DB_CC_HMI".CC_ST25_DriveRollerUp,
                         HMI_Hydraulic_Down := "DB_CC_HMI".CC_ST25_RollsDown,
                         HMI_Hydraulic_Up := "DB_CC_HMI".CC_ST25_RollsUp,
                         HMI_Modules_Down := "DB_CC_HMI".CC_ST25_ModulesDown,
                         HMI_Modules_Up := "DB_CC_HMI".CC_ST25_ModulesUp,
                         HMI_Vibrating := "DB_CC_HMI".CC_ST25_Wibrating,
                         CNT_DownPos1 := 1,
                         CNT_DownPos2 := 1,
                         CNT_UpPos1 := 1,
                         CNT_UpPos2 := 1,
                         Hydraulic_Roller_DownPos1 := "ST25_PAL_Sen12",
                         Hydraulic_Roller_DownPos2 := "ST25_PAL_Sen22",
                         Hydraulic_Roller_UpPos1 := "ST25_PAL_Sen11",
                         Hydraulic_Roller_UpPos2 := "ST25_PAL_Sen21",
                         Hydraulic_Unit_Ready := #HydraulicUnit_MC_MoveJog.InVelocity,
                         Drive_Roller_DownPos1 := "ST25_DR_a_Down",
                         Drive_Roller_DownPos2 := "ST25_DR_b_Down",
                         Drive_Roller_UpPos1 := "ST25_DR_a_Up",
                         Drive_Roller_UpPos2 := "ST25_DR_b_Up",
                         Modules_DownPos1 := "ST25_MOD1_Sen11" AND "ST25_MOD2_Sen11" AND "ST25_MOD3_Sen11",
                         Modules_DownPos2 := "ST25_MOD1_Sen21" AND "ST25_MOD2_Sen21" AND "ST25_MOD3_Sen21",
                         Modules_UpPos1 := "ST25_MOD1_Sen12" AND "ST25_MOD2_Sen12" AND "ST25_MOD3_Sen12",
                         Modules_UpPos2 := "ST25_MOD1_Sen22" AND "ST25_MOD2_Sen22" AND "ST25_MOD3_Sen22",
                         Hydraulic_Unit => #ST25_Station_Control.Hydraulic_Unit,
                         Hydraulic_Rollers_Up => "ST25_Hydraulic_Rollers_Up",
                         Hydraulic_Rollers_Down => "ST25_Hydraulic_Rollers_Down",
                         Vibration_Enable => #ST25_Station_Control.Vibration_Enable,
                         Drive_Rollers_Up => "ST25_Drivers_Rollers_Up",
                         Modules_Up => "ST25_Modules_Up");
END_REGION

REGION Network 4: Data to safety set hydraulic main valve
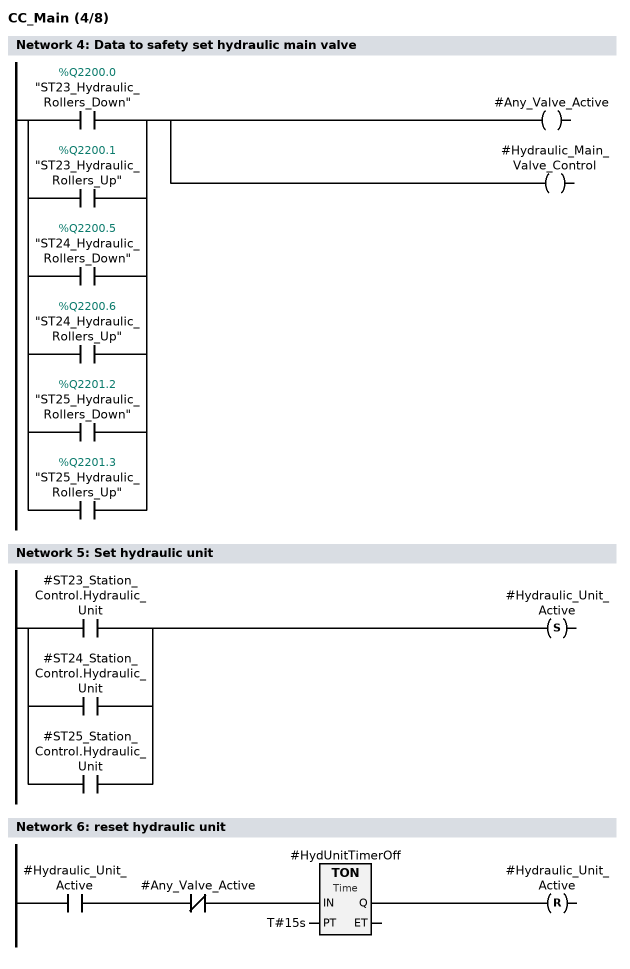
   RUNG wire#powerrail
      Contact( "ST23_Hydraulic_Rollers_Down" )
      wire#w1
      Coil( #Any_Valve_Active )
   END_RUNG
   RUNG wire#powerrail
      Contact( "ST23_Hydraulic_Rollers_Up" )
   END_RUNG wire#w1
   RUNG wire#powerrail
      Contact( "ST24_Hydraulic_Rollers_Down" )
   END_RUNG wire#w1
   RUNG wire#powerrail
      Contact( "ST24_Hydraulic_Rollers_Up" )
   END_RUNG wire#w1
   RUNG wire#powerrail
      Contact( "ST25_Hydraulic_Rollers_Down" )
   END_RUNG wire#w1
   RUNG wire#powerrail
      Contact( "ST25_Hydraulic_Rollers_Up" )
   END_RUNG wire#w1
   RUNG wire#w1
      Coil( #Hydraulic_Main_Valve_Control )
   END_RUNG
   // the same network as SCL:
   #Any_Valve_Active := "ST23_Hydraulic_Rollers_Down" OR "ST23_Hydraulic_Rollers_Up" OR "ST24_Hydraulic_Rollers_Down" OR "ST24_Hydraulic_Rollers_Up" OR "ST25_Hydraulic_Rollers_Down" OR "ST25_Hydraulic_Rollers_Up";
   #Hydraulic_Main_Valve_Control := #Any_Valve_Active;
END_REGION

REGION Network 5: Set hydraulic unit
   RUNG wire#powerrail
      Contact( #ST23_Station_Control.Hydraulic_Unit )
      wire#w1
      S_Coil( #Hydraulic_Unit_Active )
   END_RUNG
   RUNG wire#powerrail
      Contact( #ST24_Station_Control.Hydraulic_Unit )
   END_RUNG wire#w1
   RUNG wire#powerrail
      Contact( #ST25_Station_Control.Hydraulic_Unit )
   END_RUNG wire#w1
   // the same network as SCL:
   IF #ST23_Station_Control.Hydraulic_Unit OR #ST24_Station_Control.Hydraulic_Unit OR #ST25_Station_Control.Hydraulic_Unit THEN
       #Hydraulic_Unit_Active := TRUE;
   END_IF;
END_REGION

REGION Network 6: reset hydraulic unit
   RUNG wire#powerrail
      Contact( #Hydraulic_Unit_Active )
      I_Contact( #Any_Valve_Active )
      { S7_Templates := "time_type := Time" } #HydUnitTimerOff.TON(pt := T#15s, et =>)
      R_Coil( #Hydraulic_Unit_Active )
   END_RUNG
   // the same network as SCL:
   #HydUnitTimerOff(IN := #Hydraulic_Unit_Active AND NOT #Any_Valve_Active, PT := T#15s);   // TON
   IF #HydUnitTimerOff.Q THEN #Hydraulic_Unit_Active := FALSE; END_IF;
END_REGION

REGION Network 7: Hydraulic Unit Motion Control
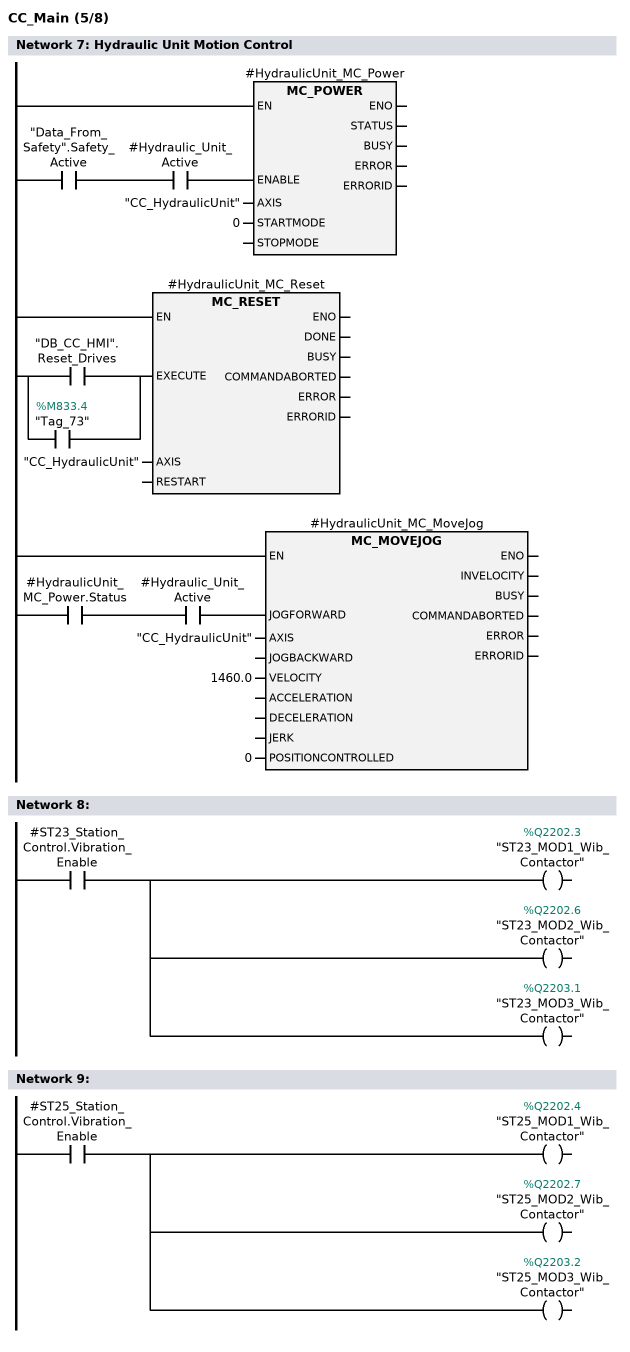
   RUNG wire#powerrail
      #HydraulicUnit_MC_Power.MC_POWER(Enable := wire#w1, Axis := "CC_HydraulicUnit", StartMode := 0, StopMode :=, Status =>, Busy =>, Error =>, ErrorId =>)
   END_RUNG
   RUNG wire#powerrail
      Contact( "Data_From_Safety".Safety_Active )
      Contact( #Hydraulic_Unit_Active )
   END_RUNG wire#w1
   RUNG wire#powerrail
      #HydraulicUnit_MC_Reset.MC_RESET(Execute := wire#w2, Axis := "CC_HydraulicUnit", Restart :=, Done =>, Busy =>, CommandAborted =>, Error =>, ErrorId =>)
   END_RUNG
   RUNG wire#powerrail
      Contact( "DB_CC_HMI".Reset_Drives )
   END_RUNG wire#w2
   RUNG wire#powerrail
      Contact( "Tag_73" )
   END_RUNG wire#w2
   RUNG wire#powerrail
      #HydraulicUnit_MC_MoveJog.MC_MOVEJOG(JogForward := wire#w3, Axis := "CC_HydraulicUnit", JogBackward :=, Velocity := 1460.0, Acceleration :=, Deceleration :=, Jerk :=, PositionControlled := 0, InVelocity =>, Busy =>, CommandAborted =>, Error =>, ErrorId =>)
   END_RUNG
   RUNG wire#powerrail
      Contact( #HydraulicUnit_MC_Power.Status )
      Contact( #Hydraulic_Unit_Active )
   END_RUNG wire#w3
   // the same network as SCL:
   #HydraulicUnit_MC_Power(Enable := "Data_From_Safety".Safety_Active AND #Hydraulic_Unit_Active,   // MC_POWER
                           Axis := "CC_HydraulicUnit",
                           StartMode := 0);
   #HydraulicUnit_MC_Reset(Execute := "DB_CC_HMI".Reset_Drives OR "Tag_73", Axis := "CC_HydraulicUnit");   // MC_RESET
   #HydraulicUnit_MC_MoveJog(JogForward := #HydraulicUnit_MC_Power.Status AND #Hydraulic_Unit_Active,   // MC_MOVEJOG
                           Axis := "CC_HydraulicUnit",
                           Velocity := 1460.0,
                           PositionControlled := 0);
END_REGION

REGION Network 8
   RUNG wire#powerrail
      Contact( #ST23_Station_Control.Vibration_Enable )
      wire#w1
      Coil( "ST23_MOD1_Wib_Contactor" )
   END_RUNG
   RUNG wire#w1
      Coil( "ST23_MOD2_Wib_Contactor" )
   END_RUNG
   RUNG wire#w1
      Coil( "ST23_MOD3_Wib_Contactor" )
   END_RUNG
   // the same network as SCL:
   "ST23_MOD1_Wib_Contactor" := #ST23_Station_Control.Vibration_Enable;
   "ST23_MOD2_Wib_Contactor" := #ST23_Station_Control.Vibration_Enable;
   "ST23_MOD3_Wib_Contactor" := #ST23_Station_Control.Vibration_Enable;
END_REGION

REGION Network 9
   RUNG wire#powerrail
      Contact( #ST25_Station_Control.Vibration_Enable )
      wire#w1
      Coil( "ST25_MOD1_Wib_Contactor" )
   END_RUNG
   RUNG wire#w1
      Coil( "ST25_MOD2_Wib_Contactor" )
   END_RUNG
   RUNG wire#w1
      Coil( "ST25_MOD3_Wib_Contactor" )
   END_RUNG
   // the same network as SCL:
   "ST25_MOD1_Wib_Contactor" := #ST25_Station_Control.Vibration_Enable;
   "ST25_MOD2_Wib_Contactor" := #ST25_Station_Control.Vibration_Enable;
   "ST25_MOD3_Wib_Contactor" := #ST25_Station_Control.Vibration_Enable;
END_REGION

REGION Network 10
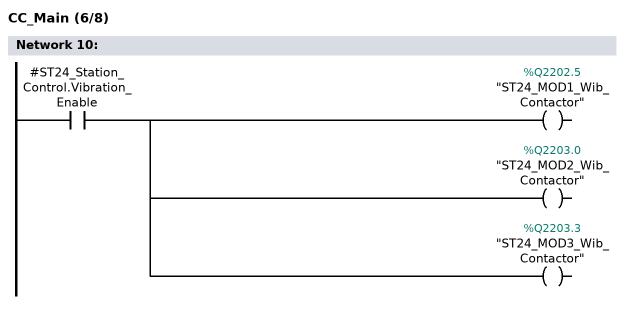
   RUNG wire#powerrail
      Contact( #ST24_Station_Control.Vibration_Enable )
      wire#w1
      Coil( "ST24_MOD1_Wib_Contactor" )
   END_RUNG
   RUNG wire#w1
      Coil( "ST24_MOD2_Wib_Contactor" )
   END_RUNG
   RUNG wire#w1
      Coil( "ST24_MOD3_Wib_Contactor" )
   END_RUNG
   // the same network as SCL:
   "ST24_MOD1_Wib_Contactor" := #ST24_Station_Control.Vibration_Enable;
   "ST24_MOD2_Wib_Contactor" := #ST24_Station_Control.Vibration_Enable;
   "ST24_MOD3_Wib_Contactor" := #ST24_Station_Control.Vibration_Enable;
END_REGION

REGION Network 11
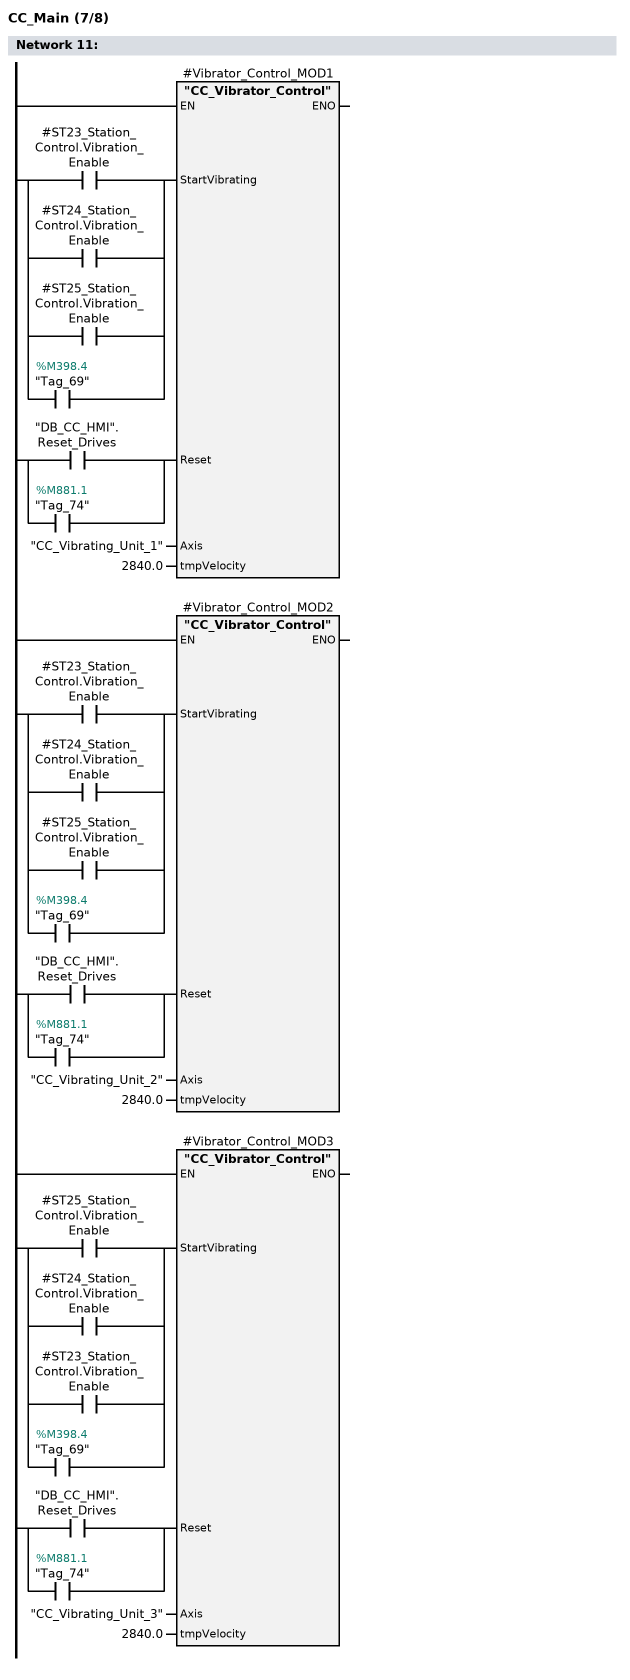
   RUNG wire#powerrail
      #Vibrator_Control_MOD1(StartVibrating := wire#w1, Reset := wire#w2, Axis := "CC_Vibrating_Unit_1", tmpVelocity := 2840.0)
   END_RUNG
   RUNG wire#powerrail
      Contact( #ST23_Station_Control.Vibration_Enable )
   END_RUNG wire#w1
   RUNG wire#powerrail
      Contact( #ST24_Station_Control.Vibration_Enable )
   END_RUNG wire#w1
   RUNG wire#powerrail
      Contact( #ST25_Station_Control.Vibration_Enable )
   END_RUNG wire#w1
   RUNG wire#powerrail
      Contact( "Tag_69" )
   END_RUNG wire#w1
   RUNG wire#powerrail
      Contact( "DB_CC_HMI".Reset_Drives )
   END_RUNG wire#w2
   RUNG wire#powerrail
      Contact( "Tag_74" )
   END_RUNG wire#w2
   RUNG wire#powerrail
      #Vibrator_Control_MOD2(StartVibrating := wire#w3, Reset := wire#w4, Axis := "CC_Vibrating_Unit_2", tmpVelocity := 2840.0)
   END_RUNG
   RUNG wire#powerrail
      Contact( #ST23_Station_Control.Vibration_Enable )
   END_RUNG wire#w3
   RUNG wire#powerrail
      Contact( #ST24_Station_Control.Vibration_Enable )
   END_RUNG wire#w3
   RUNG wire#powerrail
      Contact( #ST25_Station_Control.Vibration_Enable )
   END_RUNG wire#w3
   RUNG wire#powerrail
      Contact( "Tag_69" )
   END_RUNG wire#w3
   RUNG wire#powerrail
      Contact( "DB_CC_HMI".Reset_Drives )
   END_RUNG wire#w4
   RUNG wire#powerrail
      Contact( "Tag_74" )
   END_RUNG wire#w4
   RUNG wire#powerrail
      #Vibrator_Control_MOD3(StartVibrating := wire#w5, Reset := wire#w6, Axis := "CC_Vibrating_Unit_3", tmpVelocity := 2840.0)
   END_RUNG
   RUNG wire#powerrail
      Contact( #ST25_Station_Control.Vibration_Enable )
   END_RUNG wire#w5
   RUNG wire#powerrail
      Contact( #ST24_Station_Control.Vibration_Enable )
   END_RUNG wire#w5
   RUNG wire#powerrail
      Contact( #ST23_Station_Control.Vibration_Enable )
   END_RUNG wire#w5
   RUNG wire#powerrail
      Contact( "Tag_69" )
   END_RUNG wire#w5
   RUNG wire#powerrail
      Contact( "DB_CC_HMI".Reset_Drives )
   END_RUNG wire#w6
   RUNG wire#powerrail
      Contact( "Tag_74" )
   END_RUNG wire#w6
   // the same network as SCL:
   #Vibrator_Control_MOD1(StartVibrating := #ST23_Station_Control.Vibration_Enable OR #ST24_Station_Control.Vibration_Enable OR #ST25_Station_Control.Vibration_Enable OR "Tag_69",   // "CC_Vibrator_Control"
                          Reset := "DB_CC_HMI".Reset_Drives OR "Tag_74",
                          Axis := "CC_Vibrating_Unit_1",
                          tmpVelocity := 2840.0);
   #Vibrator_Control_MOD2(StartVibrating := #ST23_Station_Control.Vibration_Enable OR #ST24_Station_Control.Vibration_Enable OR #ST25_Station_Control.Vibration_Enable OR "Tag_69",   // "CC_Vibrator_Control"
                          Reset := "DB_CC_HMI".Reset_Drives OR "Tag_74",
                          Axis := "CC_Vibrating_Unit_2",
                          tmpVelocity := 2840.0);
   #Vibrator_Control_MOD3(StartVibrating := #ST25_Station_Control.Vibration_Enable OR #ST24_Station_Control.Vibration_Enable OR #ST23_Station_Control.Vibration_Enable OR "Tag_69",   // "CC_Vibrator_Control"
                          Reset := "DB_CC_HMI".Reset_Drives OR "Tag_74",
                          Axis := "CC_Vibrating_Unit_3",
                          tmpVelocity := 2840.0);
END_REGION

REGION Network 12
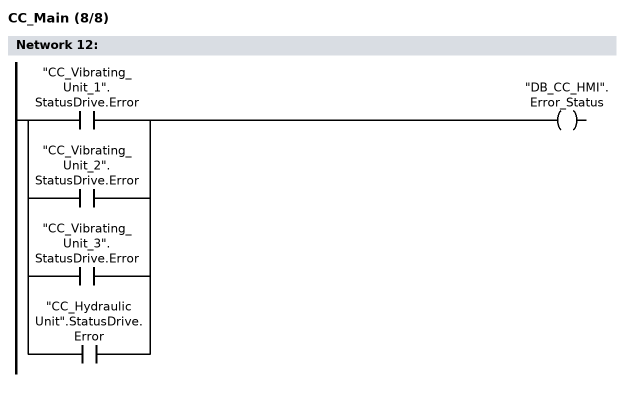
   RUNG wire#powerrail
      Contact( "CC_Vibrating_Unit_1".StatusDrive.Error )
      wire#w1
      Coil( "DB_CC_HMI".Error_Status )
   END_RUNG
   RUNG wire#powerrail
      Contact( "CC_Vibrating_Unit_2".StatusDrive.Error )
   END_RUNG wire#w1
   RUNG wire#powerrail
      Contact( "CC_Vibrating_Unit_3".StatusDrive.Error )
   END_RUNG wire#w1
   RUNG wire#powerrail
      Contact( "CC_HydraulicUnit".StatusDrive.Error )
   END_RUNG wire#w1
   // the same network as SCL:
   "DB_CC_HMI".Error_Status := "CC_Vibrating_Unit_1".StatusDrive.Error OR "CC_Vibrating_Unit_2".StatusDrive.Error OR "CC_Vibrating_Unit_3".StatusDrive.Error OR "CC_HydraulicUnit".StatusDrive.Error;
END_REGION
END_FUNCTION_BLOCK

FUNCTION_BLOCK "CC_Station_Control"   // FB105, LAD
{ S7_Optimized_Access := 'TRUE' }
// stored: AutoNumber false, MemoryReserve 100, SetENOAutomatically false
   VAR_INPUT
      HMI_Reset : Bool;
      Station_Empty : Bool;
      Station_Occupied : Bool;
      Button_Seq_Forward : Bool;
      Button_Seq_Backward : Bool;
      HMI_Drive_Rollers_Down : Bool;
      HMI_Drive_Rollers_Up : Bool;
      HMI_Hydraulic_Down : Bool;
      HMI_Hydraulic_Up : Bool;
      HMI_Modules_Down : Bool;
      HMI_Modules_Up : Bool;
      HMI_Vibrating : Bool;
      CNT_DownPos1 : Bool;
      CNT_DownPos2 : Bool;
      CNT_UpPos1 : Bool;
      CNT_UpPos2 : Bool;
      Hydraulic_Roller_DownPos1 : Bool;
      Hydraulic_Roller_DownPos2 : Bool;
      Hydraulic_Roller_UpPos1 : Bool;
      Hydraulic_Roller_UpPos2 : Bool;
      Hydraulic_Unit_Ready : Bool;
      Drive_Roller_DownPos1 : Bool;
      Drive_Roller_DownPos2 : Bool;
      Drive_Roller_UpPos1 : Bool;
      Drive_Roller_UpPos2 : Bool;
      Modules_DownPos1 : Bool;
      Modules_DownPos2 : Bool;
      Modules_UpPos1 : Bool;
      Modules_UpPos2 : Bool;
   END_VAR
   VAR_OUTPUT
      Hydraulic_Unit : Bool;
      Hydraulic_Rollers_Up : Bool;
      Hydraulic_Rollers_Down : Bool;
      Vibration_Enable : Bool;
      Drive_Rollers_Up : Bool;
      Modules_Up : Bool;
   END_VAR
   VAR
      Hydraulic_Unit_Active : Bool;
      Hydraulic_Unit_TimerOff { S7_SetPoint := 'True'} : TON_TIME;
      Hydraulic_Unit_MC_Power { S7_SetPoint := 'True'} : MC_POWER;
      Hydraulic_Rollers { S7_SetPoint := 'True'} : "CC_Hydraulic_Rollers";
      Pneumatic_Rollers { S7_SetPoint := 'True'} : "CC_Pneumatic_Roller";
      Vibrator_Control { S7_SetPoint := 'True'} : "CC_Vibrator_Control";
      Sequence_Step { S7_SetPoint := 'True'} : Int;
      Req_Hydraulic_Rollers_Up : Bool;
      Req_Hydraulic_Rollers_Down : Bool;
      Req_Drive_Roller_Up : Bool;
      Req_Drive_Roller_Down : Bool;
      Req_Vibration_Enable : Bool;
      Req_Modules_Up : Bool;
      Req_Modules_Down : Bool;
      Sequence_Control { S7_SetPoint := 'True'} : "CC_Sequence_Control";
      Module_Control { S7_SetPoint := 'True'} : "CC_Vib_Modules";
      Hyd_Rollers_Up_whenMoving { S7_SetPoint := 'True'} : Bool;
   END_VAR
BEGIN

REGION Network 1: Centering devices position down
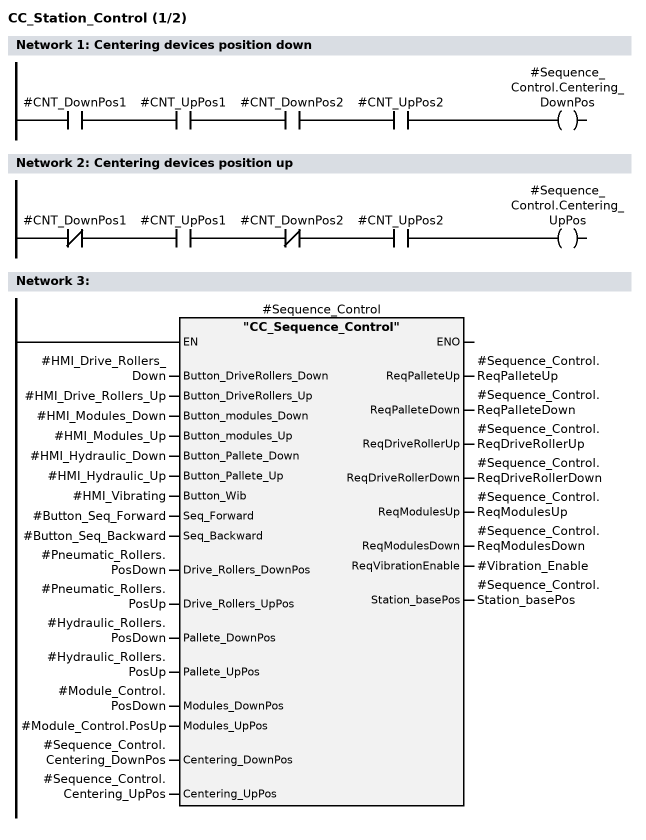
   RUNG wire#powerrail
      Contact( #CNT_DownPos1 )
      Contact( #CNT_UpPos1 )
      Contact( #CNT_DownPos2 )
      Contact( #CNT_UpPos2 )
      Coil( #Sequence_Control.Centering_DownPos )
   END_RUNG
   // the same network as SCL:
   #Sequence_Control.Centering_DownPos := #CNT_DownPos1 AND #CNT_UpPos1 AND #CNT_DownPos2 AND #CNT_UpPos2;
END_REGION

REGION Network 2: Centering devices position up
   RUNG wire#powerrail
      I_Contact( #CNT_DownPos1 )
      Contact( #CNT_UpPos1 )
      I_Contact( #CNT_DownPos2 )
      Contact( #CNT_UpPos2 )
      Coil( #Sequence_Control.Centering_UpPos )
   END_RUNG
   // the same network as SCL:
   #Sequence_Control.Centering_UpPos := NOT #CNT_DownPos1 AND #CNT_UpPos1 AND NOT #CNT_DownPos2 AND #CNT_UpPos2;
END_REGION

REGION Network 3
   RUNG wire#powerrail
      #Sequence_Control(Button_DriveRollers_Down := #HMI_Drive_Rollers_Down, Button_DriveRollers_Up := #HMI_Drive_Rollers_Up, Button_modules_Down := #HMI_Modules_Down, Button_modules_Up := #HMI_Modules_Up, Button_Pallete_Down := #HMI_Hydraulic_Down, Button_Pallete_Up := #HMI_Hydraulic_Up, Button_Wib := #HMI_Vibrating, Seq_Forward := #Button_Seq_Forward, Seq_Backward := #Button_Seq_Backward, Drive_Rollers_DownPos := #Pneumatic_Rollers.PosDown, Drive_Rollers_UpPos := #Pneumatic_Rollers.PosUp, Pallete_DownPos := #Hydraulic_Rollers.PosDown, Pallete_UpPos := #Hydraulic_Rollers.PosUp, Modules_DownPos := #Module_Control.PosDown, Modules_UpPos := #Module_Control.PosUp, Centering_DownPos := #Sequence_Control.Centering_DownPos, Centering_UpPos := #Sequence_Control.Centering_UpPos, ReqPalleteUp => #Sequence_Control.ReqPalleteUp, ReqPalleteDown => #Sequence_Control.ReqPalleteDown, ReqDriveRollerUp => #Sequence_Control.ReqDriveRollerUp, ReqDriveRollerDown => #Sequence_Control.ReqDriveRollerDown, ReqModulesUp => #Sequence_Control.ReqModulesUp, ReqModulesDown => #Sequence_Control.ReqModulesDown, ReqVibrationEnable => #Vibration_Enable, Station_basePos => #Sequence_Control.Station_basePos)
   END_RUNG
   // the same network as SCL:
   #Sequence_Control(Button_DriveRollers_Down := #HMI_Drive_Rollers_Down,   // "CC_Sequence_Control"
                     Button_DriveRollers_Up := #HMI_Drive_Rollers_Up,
                     Button_modules_Down := #HMI_Modules_Down,
                     Button_modules_Up := #HMI_Modules_Up,
                     Button_Pallete_Down := #HMI_Hydraulic_Down,
                     Button_Pallete_Up := #HMI_Hydraulic_Up,
                     Button_Wib := #HMI_Vibrating,
                     Seq_Forward := #Button_Seq_Forward,
                     Seq_Backward := #Button_Seq_Backward,
                     Drive_Rollers_DownPos := #Pneumatic_Rollers.PosDown,
                     Drive_Rollers_UpPos := #Pneumatic_Rollers.PosUp,
                     Pallete_DownPos := #Hydraulic_Rollers.PosDown,
                     Pallete_UpPos := #Hydraulic_Rollers.PosUp,
                     Modules_DownPos := #Module_Control.PosDown,
                     Modules_UpPos := #Module_Control.PosUp,
                     Centering_DownPos := #Sequence_Control.Centering_DownPos,
                     Centering_UpPos := #Sequence_Control.Centering_UpPos,
                     ReqPalleteUp => #Sequence_Control.ReqPalleteUp,
                     ReqPalleteDown => #Sequence_Control.ReqPalleteDown,
                     ReqDriveRollerUp => #Sequence_Control.ReqDriveRollerUp,
                     ReqDriveRollerDown => #Sequence_Control.ReqDriveRollerDown,
                     ReqModulesUp => #Sequence_Control.ReqModulesUp,
                     ReqModulesDown => #Sequence_Control.ReqModulesDown,
                     ReqVibrationEnable => #Vibration_Enable,
                     Station_basePos => #Sequence_Control.Station_basePos);
END_REGION

REGION Network 4: Hydraulic rollers control
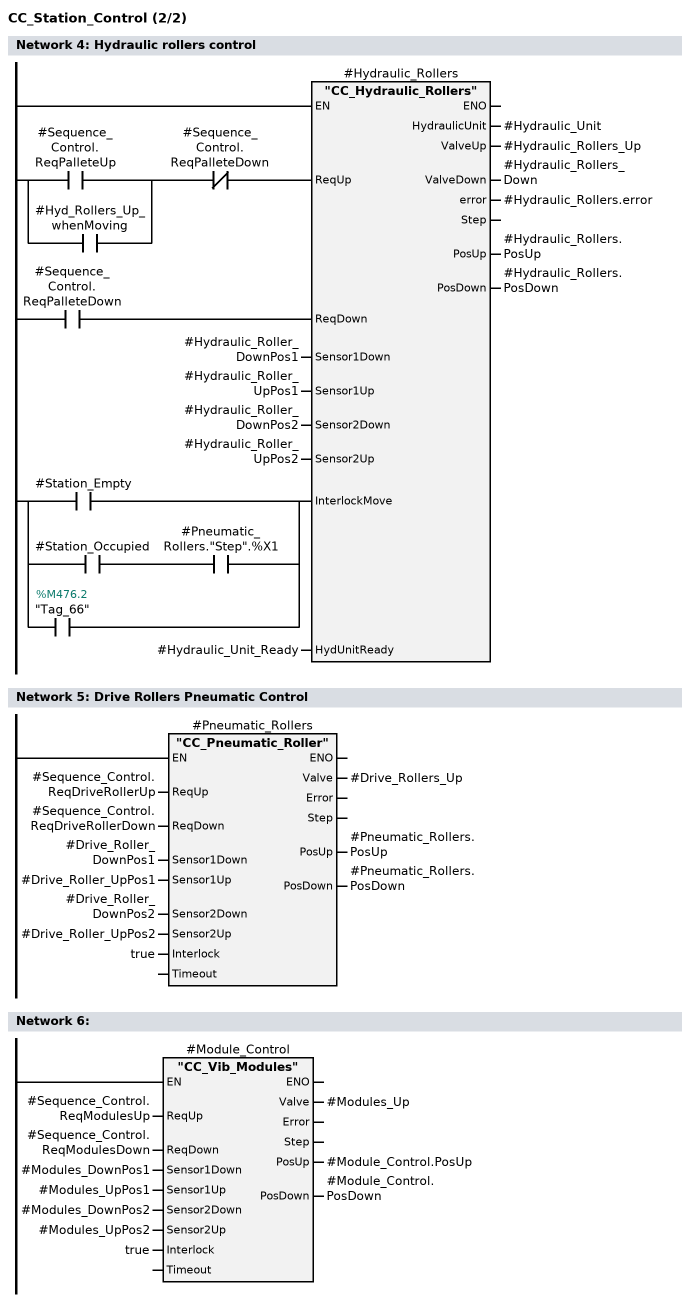
   RUNG wire#powerrail
      #Hydraulic_Rollers(ReqUp := wire#w2, ReqDown := wire#w3, InterlockMove := wire#w4, Sensor1Down := #Hydraulic_Roller_DownPos1, Sensor1Up := #Hydraulic_Roller_UpPos1, Sensor2Down := #Hydraulic_Roller_DownPos2, Sensor2Up := #Hydraulic_Roller_UpPos2, HydUnitReady := #Hydraulic_Unit_Ready, HydraulicUnit => #Hydraulic_Unit, ValveUp => #Hydraulic_Rollers_Up, ValveDown => #Hydraulic_Rollers_Down, error => #Hydraulic_Rollers.error, "Step" =>, PosUp => #Hydraulic_Rollers.PosUp, PosDown => #Hydraulic_Rollers.PosDown)
   END_RUNG
   RUNG wire#powerrail
      Contact( #Sequence_Control.ReqPalleteUp )
      wire#w1
      I_Contact( #Sequence_Control.ReqPalleteDown )
   END_RUNG wire#w2
   RUNG wire#powerrail
      Contact( #Hyd_Rollers_Up_whenMoving )
   END_RUNG wire#w1
   RUNG wire#powerrail
      Contact( #Sequence_Control.ReqPalleteDown )
   END_RUNG wire#w3
   RUNG wire#powerrail
      Contact( #Station_Empty )
   END_RUNG wire#w4
   RUNG wire#powerrail
      Contact( #Station_Occupied )
      Contact( #Pneumatic_Rollers."Step".%X1 )
   END_RUNG wire#w4
   RUNG wire#powerrail
      Contact( "Tag_66" )
   END_RUNG wire#w4
   // the same network as SCL:
   #Hydraulic_Rollers(ReqUp := (#Sequence_Control.ReqPalleteUp OR #Hyd_Rollers_Up_whenMoving) AND NOT #Sequence_Control.ReqPalleteDown,   // "CC_Hydraulic_Rollers"
                      ReqDown := #Sequence_Control.ReqPalleteDown,
                      Sensor1Down := #Hydraulic_Roller_DownPos1,
                      Sensor1Up := #Hydraulic_Roller_UpPos1,
                      Sensor2Down := #Hydraulic_Roller_DownPos2,
                      Sensor2Up := #Hydraulic_Roller_UpPos2,
                      InterlockMove := #Station_Empty OR (#Station_Occupied AND #Pneumatic_Rollers."Step".%X1) OR "Tag_66",
                      HydUnitReady := #Hydraulic_Unit_Ready,
                      HydraulicUnit => #Hydraulic_Unit,
                      ValveUp => #Hydraulic_Rollers_Up,
                      ValveDown => #Hydraulic_Rollers_Down,
                      error => #Hydraulic_Rollers.error,
                      PosUp => #Hydraulic_Rollers.PosUp,
                      PosDown => #Hydraulic_Rollers.PosDown);
END_REGION

REGION Network 5: Drive Rollers Pneumatic Control
   RUNG wire#powerrail
      #Pneumatic_Rollers(ReqUp := #Sequence_Control.ReqDriveRollerUp, ReqDown := #Sequence_Control.ReqDriveRollerDown, Sensor1Down := #Drive_Roller_DownPos1, Sensor1Up := #Drive_Roller_UpPos1, Sensor2Down := #Drive_Roller_DownPos2, Sensor2Up := #Drive_Roller_UpPos2, Interlock := true, Timeout :=, Valve => #Drive_Rollers_Up, Error =>, "Step" =>, PosUp => #Pneumatic_Rollers.PosUp, PosDown => #Pneumatic_Rollers.PosDown)
   END_RUNG
   // the same network as SCL:
   #Pneumatic_Rollers(ReqUp := #Sequence_Control.ReqDriveRollerUp,   // "CC_Pneumatic_Roller"
                      ReqDown := #Sequence_Control.ReqDriveRollerDown,
                      Sensor1Down := #Drive_Roller_DownPos1,
                      Sensor1Up := #Drive_Roller_UpPos1,
                      Sensor2Down := #Drive_Roller_DownPos2,
                      Sensor2Up := #Drive_Roller_UpPos2,
                      Interlock := true,
                      Valve => #Drive_Rollers_Up,
                      PosUp => #Pneumatic_Rollers.PosUp,
                      PosDown => #Pneumatic_Rollers.PosDown);
END_REGION

